C03624=1096.726,72.029,-58.754,176.200,16.216,152.221
C03625=1096.720,71.780,-58.738,176.198,16.216,152.221
C03626=1096.715,71.531,-58.720,176.195,16.215,152.221
C03627=1096.709,71.282,-58.704,176.193,16.214,152.222
C03628=1096.703,71.032,-58.687,176.190,16.213,152.222
C03629=1096.698,70.783,-58.670,176.188,16.213,152.222
C03630=1096.692,70.534,-58.654,176.185,16.211,152.223
C03631=1096.687,70.284,-58.637,176.183,16.211,152.223
C03632=1096.681,70.035,-58.620,176.180,16.210,152.223
C03633=1096.675,69.785,-58.602,176.179,16.209,152.224
C03634=1096.669,69.536,-58.586,176.176,16.209,152.224
C03635=1096.663,69.286,-58.569,176.174,16.208,152.224
C03636=1096.657,69.037,-58.552,176.172,16.207,152.225
C03637=1096.652,68.787,-58.536,176.169,16.206,152.225
C03638=1096.646,68.538,-58.519,176.167,16.205,152.225
C03639=1096.641,68.288,-58.502,176.164,16.205,152.226
C03640=1096.635,68.039,-58.486,176.162,16.204,152.226
C03641=1096.629,67.790,-58.469,176.159,16.203,152.226
C03642=1096.623,67.541,-58.452,176.157,16.202,152.227
C03643=1096.618,67.291,-58.436,176.155,16.201,152.227
C03644=1096.612,67.042,-58.419,176.152,16.201,152.227
C03645=1096.606,66.793,-58.402,176.150,16.200,152.228
C03646=1096.601,66.543,-58.385,176.148,16.199,152.228
C03647=1096.595,66.294,-58.369,176.146,16.199,152.228
C03648=1096.590,66.044,-58.352,176.143,16.197,152.228
C03649=1096.584,65.795,-58.336,176.141,16.197,152.229
C03650=1096.578,65.546,-58.320,176.138,16.196,152.229
C03651=1096.572,65.296,-58.303,176.136,16.195,152.229
C03652=1096.566,65.047,-58.286,176.133,16.194,152.230
C03653=1096.561,64.798,-58.269,176.131,16.194,152.230
C03654=1096.555,64.548,-58.253,176.129,16.192,152.230
C03655=1096.549,64.299,-58.237,176.127,16.192,152.231
C03656=1096.543,64.024,-58.218,176.124,16.191,152.231
C03657=1096.537,63.749,-58.200,176.122,16.190,152.231
C03658=1096.531,63.475,-58.182,176.119,16.189,152.232
C03659=1096.524,63.201,-58.164,176.116,16.188,152.232
C03660=1096.519,62.952,-58.147,176.114,16.187,152.232
C03661=1096.513,62.702,-58.131,176.111,16.186,152.233
C03662=1096.507,62.453,-58.115,176.109,16.186,152.233
C03663=1096.501,62.204,-58.098,176.107,16.185,152.233
C03664=1096.495,61.954,-58.082,176.105,16.184,152.234
C03665=1096.490,61.705,-58.065,176.103,16.184,152.234
C03666=1096.484,61.455,-58.049,176.100,16.182,152.234
C03667=1096.478,61.206,-58.033,176.098,16.182,152.235
C03668=1096.472,60.957,-58.017,176.095,16.181,152.235
C03669=1096.466,60.707,-58.000,176.093,16.180,152.235
C03670=1096.461,60.458,-57.983,176.091,16.179,152.235
C03671=1096.455,60.208,-57.967,176.088,16.179,152.236
C03672=1096.449,59.959,-57.951,176.086,16.178,152.236
C03673=1096.443,59.709,-57.935,176.084,16.177,152.236
C03674=1096.437,59.460,-57.918,176.082,16.176,152.237
C03675=1096.432,59.210,-57.902,176.079,16.175,152.237
C03676=1096.426,58.961,-57.885,176.077,16.174,152.237
C03677=1096.420,58.711,-57.870,176.075,16.174,152.238
C03678=1096.414,58.462,-57.854,176.072,16.172,152.238
C03679=1096.408,58.212,-57.837,176.070,16.172,152.238
C03680=1096.403,57.964,-57.821,176.068,16.171,152.239
C03681=1096.397,57.714,-57.805,176.066,16.170,152.239
C03682=1096.391,57.465,-57.788,176.063,16.169,152.239
C03683=1096.386,57.215,-57.772,176.061,16.168,152.239
C03684=1096.380,56.966,-57.756,176.059,16.168,152.240
C03685=1096.374,56.716,-57.740,176.056,16.167,152.240
C03686=1096.368,56.467,-57.724,176.054,16.166,152.240
C03687=1096.362,56.217,-57.708,176.052,16.165,152.240
C03688=1096.356,55.968,-57.691,176.050,16.164,152.241
C03689=1096.351,55.719,-57.675,176.048,16.163,152.241
C03690=1096.346,55.469,-57.659,176.045,16.162,152.241
C03691=1096.340,55.220,-57.643,176.043,16.161,152.242
C03692=1096.334,54.970,-57.627,176.040,16.161,152.242
C03693=1096.328,54.721,-57.611,176.038,16.160,152.242
C03694=1096.322,54.472,-57.594,176.036,16.159,152.242
C03695=1096.317,54.223,-57.579,176.034,16.158,152.243
C03696=1096.311,53.973,-57.563,176.032,16.157,152.243
C03697=1096.305,53.724,-57.547,176.029,16.156,152.243
C03698=1096.299,53.474,-57.531,176.027,16.155,152.244
C03699=1096.294,53.224,-57.514,176.025,16.154,152.244
C03700=1096.288,52.975,-57.498,176.023,16.153,152.244
C03701=1096.283,52.726,-57.482,176.021,16.153,152.244
C03702=1096.277,52.476,-57.467,176.018,16.151,152.245
C03703=1096.271,52.227,-57.450,176.016,16.151,152.245
C03704=1096.265,51.978,-57.434,176.014,16.149,152.245
C03705=1096.260,51.728,-57.419,176.011,16.149,152.246
C03706=1096.254,51.479,-57.403,176.010,16.148,152.246
C03707=1096.248,51.230,-57.386,176.007,16.147,152.246
C03708=1096.243,50.980,-57.371,176.005,16.146,152.246
C03709=1096.237,50.730,-57.355,176.002,16.145,152.247
C03710=1096.232,50.481,-57.339,176.000,16.144,152.247
C03711=1096.226,50.232,-57.323,175.999,16.144,152.247
C03712=1096.220,49.982,-57.307,175.996,16.142,152.247
C03713=1096.214,49.732,-57.291,175.994,16.142,152.248
C03714=1096.209,49.484,-57.276,175.991,16.140,152.248
C03715=1096.203,49.234,-57.260,175.989,16.140,152.248
C03716=1096.197,48.984,-57.244,175.988,16.139,152.248
C03717=1096.191,48.735,-57.227,175.985,16.137,152.249
C03718=1096.186,48.486,-57.212,175.983,16.137,152.249
C03719=1096.180,48.236,-57.196,175.981,16.135,152.249
C03720=1096.174,47.961,-57.178,175.979,16.135,152.249
C03721=1096.168,47.687,-57.161,175.976,16.133,152.250
C03722=1096.162,47.412,-57.143,175.973,16.132,152.250
C03723=1096.156,47.138,-57.127,175.971,16.131,152.250
C03724=1096.150,46.888,-57.111,175.969,16.130,152.250
C03725=1096.144,46.639,-57.095,175.967,16.129,152.251
C03726=1096.139,46.389,-57.079,175.965,16.129,152.251
C03727=1096.134,46.139,-57.064,175.962,16.127,152.251
C03728=1096.128,45.890,-57.048,175.960,16.127,152.251
C03729=1096.122,45.640,-57.032,175.958,16.125,152.252
C03730=1096.117,45.391,-57.016,175.956,16.125,152.252
C03731=1096.111,45.141,-57.001,175.954,16.124,152.252
C03732=1096.105,44.892,-56.985,175.951,16.122,152.252
C03733=1096.100,44.643,-56.969,175.950,16.122,152.253
C03734=1096.094,44.393,-56.953,175.948,16.121,152.253
C03735=1096.089,44.144,-56.938,175.945,16.120,152.253
C03736=1096.083,43.894,-56.922,175.943,16.119,152.253
C03737=1096.077,43.645,-56.906,175.940,16.118,152.254
C03738=1096.072,43.396,-56.891,175.939,16.117,152.254
C03739=1096.066,43.146,-56.876,175.937,16.116,152.254
C03740=1096.060,42.897,-56.860,175.934,16.115,152.254
C03741=1096.055,42.647,-56.845,175.932,16.114,152.255
C03742=1096.049,42.398,-56.828,175.930,16.112,152.255
C03743=1096.043,42.148,-56.813,175.928,16.112,152.255
C03744=1096.038,41.899,-56.798,175.926,16.111,152.255
C03745=1096.032,41.650,-56.782,175.923,16.110,152.256
C03746=1096.026,41.400,-56.766,175.921,16.109,152.256
C03747=1096.021,41.151,-56.751,175.919,16.108,152.256
C03748=1096.015,40.901,-56.736,175.917,16.107,152.256
C03749=1096.009,40.651,-56.720,175.915,16.106,152.256
C03750=1096.004,40.402,-56.705,175.913,16.105,152.257
C03751=1095.998,40.152,-56.689,175.911,16.104,152.257
C03752=1095.991,39.903,-56.674,175.909,16.103,152.257
C03753=1095.986,39.654,-56.658,175.906,16.102,152.258
C03754=1095.981,39.404,-56.643,175.904,16.101,152.258
C03755=1095.975,39.155,-56.628,175.903,16.100,152.258
C03756=1095.969,38.906,-56.612,175.900,16.099,152.258
C03757=1095.963,38.656,-56.597,175.898,16.098,152.258
C03758=1095.958,38.406,-56.581,175.896,16.098,152.259
C03759=1095.952,38.157,-56.566,175.893,16.096,152.259
C03760=1095.947,37.908,-56.551,175.892,16.095,152.259
C03761=1095.941,37.658,-56.535,175.890,16.094,152.259
C03762=1095.934,37.409,-56.520,175.887,16.093,152.260
C03763=1095.929,37.159,-56.505,175.885,16.092,152.260
C03764=1095.924,36.909,-56.489,175.883,16.091,152.260
C03765=1095.918,36.660,-56.475,175.881,16.090,152.260
C03766=1095.912,36.411,-56.459,175.879,16.089,152.260
C03767=1095.906,36.161,-56.444,175.876,16.088,152.261
C03768=1095.900,35.912,-56.428,175.875,16.087,152.261
C03769=1095.894,35.662,-56.413,175.873,16.087,152.261
C03770=1095.889,35.413,-56.398,175.870,16.085,152.262
C03771=1095.883,35.163,-56.383,175.868,16.084,152.262
C03772=1095.877,34.914,-56.368,175.866,16.083,152.262
C03773=1095.872,34.664,-56.353,175.864,16.082,152.262
C03774=1095.866,34.415,-56.338,175.862,16.081,152.262
C03775=1095.860,34.166,-56.322,175.860,16.081,152.263
C03776=1095.854,33.916,-56.307,175.858,16.079,152.263
C03777=1095.849,33.667,-56.292,175.856,16.078,152.263
C03778=1095.842,33.417,-56.277,175.854,16.078,152.263
C03779=1095.837,33.167,-56.261,175.851,16.076,152.264
C03780=1095.831,32.918,-56.247,175.850,16.075,152.264
C03781=1095.825,32.668,-56.231,175.848,16.074,152.264
C03782=1095.820,32.419,-56.216,175.845,16.073,152.264
C03783=1095.814,32.170,-56.201,175.843,16.073,152.265
C03784=1095.808,31.895,-56.185,175.841,16.071,152.265
C03785=1095.802,31.621,-56.168,175.839,16.070,152.265
C03786=1095.795,31.345,-56.151,175.836,16.069,152.265
C03787=1095.789,31.071,-56.134,175.834,16.068,152.265
C03788=1095.783,30.822,-56.120,175.832,16.066,152.266
C03789=1095.778,30.572,-56.104,175.830,16.066,152.266
C03790=1095.771,30.323,-56.089,175.828,16.065,152.266
C03791=1095.766,30.073,-56.074,175.825,16.064,152.266
C03792=1095.760,29.824,-56.059,175.824,16.063,152.266
C03793=1095.755,29.574,-56.045,175.822,16.062,152.267
C03794=1095.749,29.324,-56.030,175.819,16.061,152.267
C03795=1095.744,29.075,-56.015,175.818,16.059,152.267
C03796=1095.738,28.826,-56.000,175.816,16.059,152.267
C03797=1095.732,28.576,-55.985,175.813,16.057,152.268
C03798=1095.727,28.327,-55.970,175.811,16.056,152.268
C03799=1095.720,28.077,-55.955,175.810,16.056,152.268
C03800=1095.715,27.828,-55.940,175.807,16.054,152.268
C03801=1095.709,27.578,-55.925,175.805,16.053,152.268
C03802=1095.703,27.329,-55.911,175.803,16.052,152.269
C03803=1095.698,27.079,-55.896,175.801,16.051,152.269
C03804=1095.692,26.830,-55.881,175.799,16.050,152.269
C03805=1095.686,26.580,-55.865,175.797,16.049,152.269
C03806=1095.680,26.331,-55.851,175.795,16.048,152.270
C03807=1095.674,26.081,-55.836,175.793,16.047,152.270
C03808=1095.668,25.832,-55.821,175.791,16.046,152.270
C03809=1095.663,25.582,-55.806,175.789,16.045,152.270
C03810=1095.657,25.333,-55.792,175.787,16.044,152.270
C03811=1095.651,25.083,-55.777,175.785,16.043,152.270
C03812=1095.646,24.834,-55.762,175.783,16.042,152.271
C03813=1095.640,24.584,-55.748,175.781,16.041,152.271
C03814=1095.634,24.335,-55.733,175.779,16.040,152.271
C03815=1095.629,24.085,-55.718,175.777,16.039,152.271
C03816=1095.622,23.836,-55.703,175.774,16.037,152.272
C03817=1095.617,23.586,-55.689,175.773,16.037,152.272
C03818=1095.611,23.337,-55.674,175.771,16.036,152.272
C03819=1095.605,23.087,-55.659,175.768,16.034,152.272
C03820=1095.599,22.838,-55.644,175.766,16.034,152.272
C03821=1095.594,22.588,-55.630,175.765,16.032,152.272
C03822=1095.589,22.339,-55.615,175.763,16.032,152.273
C03823=1095.582,22.089,-55.600,175.760,16.030,152.273
C03824=1095.577,21.840,-55.586,175.759,16.029,152.273
C03825=1095.570,21.590,-55.571,175.757,16.029,152.273
C03826=1095.565,21.341,-55.556,175.754,16.027,152.274
C03827=1095.560,21.091,-55.542,175.752,16.026,152.274
C03828=1095.553,20.841,-55.527,175.751,16.025,152.274
C03829=1095.548,20.592,-55.513,175.748,16.024,152.274
C03830=1095.543,20.343,-55.498,175.746,16.023,152.274
C03831=1095.537,20.093,-55.483,175.745,16.022,152.275
C03832=1095.531,19.844,-55.469,175.743,16.021,152.275
C03833=1095.525,19.594,-55.454,175.740,16.020,152.275
C03834=1095.519,19.345,-55.440,175.738,16.019,152.275
C03835=1095.513,19.095,-55.426,175.737,16.018,152.275
C03836=1095.507,18.845,-55.411,175.734,16.016,152.276
C03837=1095.502,18.596,-55.396,175.732,16.016,152.276
C03838=1095.497,18.347,-55.382,175.731,16.014,152.276
C03839=1095.490,18.097,-55.367,175.729,16.014,152.276
C03840=1095.485,17.847,-55.353,175.726,16.012,152.276
C03841=1095.479,17.598,-55.339,175.725,16.011,152.277
C03842=1095.473,17.348,-55.324,175.723,16.011,152.277
C03843=1095.467,17.099,-55.310,175.720,16.009,152.277
C03844=1095.462,16.850,-55.295,175.718,16.008,152.277
C03845=1095.456,16.600,-55.280,175.717,16.007,152.277
C03846=1095.450,16.351,-55.266,175.715,16.006,152.277
C03847=1095.445,16.101,-55.252,175.712,16.004,152.278
C03848=1095.438,15.827,-55.236,175.711,16.004,152.278
C03849=1095.431,15.554,-55.220,175.708,16.003,152.278
C03850=1095.425,15.281,-55.204,175.706,16.001,152.278
C03851=1095.419,15.008,-55.188,175.704,16.000,152.279
C03852=1095.413,14.758,-55.175,175.702,15.999,152.279
C03853=1095.408,14.509,-55.160,175.700,15.998,152.279
C03854=1095.402,14.259,-55.146,175.699,15.997,152.279
C03855=1095.396,14.010,-55.131,175.696,15.996,152.279
C03856=1095.390,13.760,-55.117,175.694,15.995,152.279
C03857=1095.384,13.511,-55.102,175.692,15.994,152.280
C03858=1095.378,13.261,-55.089,175.690,15.993,152.280
C03859=1095.373,13.012,-55.074,175.688,15.991,152.280
C03860=1095.367,12.762,-55.060,175.686,15.991,152.280
C03861=1095.361,12.512,-55.046,175.685,15.990,152.280
C03862=1095.355,12.263,-55.031,175.683,15.989,152.281
C03863=1095.349,12.013,-55.018,175.680,15.987,152.281
C03864=1095.343,11.764,-55.004,175.678,15.986,152.281
C03865=1095.337,11.515,-54.989,175.677,15.986,152.281
C03866=1095.332,11.265,-54.975,175.674,15.984,152.281
C03867=1095.325,11.015,-54.960,175.672,15.983,152.282
C03868=1095.320,10.766,-54.947,175.671,15.982,152.282
C03869=1095.314,10.516,-54.933,175.669,15.981,152.282
C03870=1095.308,10.267,-54.918,175.666,15.980,152.282
C03871=1095.303,10.017,-54.904,175.664,15.979,152.282
C03872=1095.297,9.767,-54.890,175.663,15.978,152.282
C03873=1095.291,9.519,-54.876,175.661,15.977,152.283
C03874=1095.285,9.269,-54.862,175.659,15.975,152.283
C03875=1095.279,9.019,-54.848,175.657,15.975,152.283
C03876=1095.274,8.769,-54.834,175.655,15.974,152.283
C03877=1095.268,8.520,-54.819,175.653,15.973,152.283
C03878=1095.262,8.270,-54.805,175.651,15.971,152.284
C03879=1095.256,8.021,-54.791,175.649,15.970,152.284
C03880=1095.250,7.771,-54.778,175.647,15.969,152.284
C03881=1095.244,7.522,-54.764,175.645,15.969,152.284
C03882=1095.238,7.272,-54.749,175.644,15.967,152.284
C03883=1095.233,7.023,-54.735,175.641,15.966,152.285
C03884=1095.227,6.773,-54.722,175.640,15.965,152.285
C03885=1095.221,6.524,-54.707,175.638,15.964,152.285
C03886=1095.216,6.274,-54.693,175.636,15.963,152.285
C03887=1095.209,6.024,-54.680,175.634,15.961,152.285
C03888=1095.204,5.775,-54.666,175.632,15.961,152.285
C03889=1095.198,5.525,-54.652,175.630,15.959,152.286
C03890=1095.192,5.276,-54.637,175.628,15.959,152.286
C03891=1095.187,5.027,-54.623,175.626,15.957,152.286
C03892=1095.180,4.777,-54.610,175.624,15.956,152.286
C03893=1095.175,4.527,-54.596,175.622,15.955,152.286
C03894=1095.169,4.278,-54.582,175.621,15.954,152.287
C03895=1095.164,4.028,-54.568,175.618,15.953,152.287
C03896=1095.158,3.779,-54.554,175.617,15.952,152.287
C03897=1095.152,3.529,-54.541,175.615,15.951,152.287
C03898=1095.146,3.280,-54.526,175.613,15.950,152.287
C03899=1095.140,3.030,-54.512,175.610,15.948,152.287
C03900=1095.135,2.780,-54.498,175.609,15.947,152.288
C03901=1095.129,2.531,-54.484,175.607,15.946,152.288
C03902=1095.123,2.282,-54.471,175.605,15.945,152.288
C03903=1095.118,2.032,-54.457,175.604,15.944,152.288
C03904=1095.112,1.782,-54.443,175.601,15.943,152.288
C03905=1095.106,1.532,-54.429,175.599,15.942,152.288
C03906=1095.100,1.283,-54.415,175.598,15.941,152.288
C03907=1095.094,1.033,-54.402,175.596,15.940,152.289
C03908=1095.089,0.784,-54.388,175.594,15.938,152.289
C03909=1095.083,0.534,-54.374,175.592,15.937,152.289
C03910=1095.078,0.285,-54.360,175.590,15.936,152.289
C03911=1095.072,0.035,-54.347,175.589,15.935,152.289
C03912=1095.065,-0.236,-54.332,175.586,15.934,152.290
C03913=1095.059,-0.507,-54.317,175.584,15.933,152.290
C03914=1095.053,-0.779,-54.302,175.582,15.932,152.290
C03915=1095.047,-1.049,-54.287,175.580,15.930,152.290
C03916=1095.041,-1.299,-54.273,175.578,15.929,152.290
C03917=1095.035,-1.548,-54.260,175.576,15.928,152.290
C03918=1095.029,-1.799,-54.246,175.575,15.927,152.291
C03919=1095.024,-2.048,-54.232,175.572,15.925,152.291
C03920=1095.018,-2.298,-54.219,175.571,15.925,152.291
C03921=1095.012,-2.548,-54.205,175.569,15.924,152.291
C03922=1095.007,-2.797,-54.192,175.567,15.922,152.291
C03923=1095.001,-3.047,-54.178,175.565,15.921,152.291
C03924=1094.995,-3.296,-54.164,175.563,15.920,152.292
C03925=1094.990,-3.546,-54.151,175.562,15.919,152.292
C03926=1094.984,-3.795,-54.137,175.560,15.918,152.292
C03927=1094.978,-4.044,-54.123,175.558,15.917,152.292
C03928=1094.972,-4.294,-54.110,175.555,15.916,152.292
C03929=1094.966,-4.543,-54.096,175.554,15.915,152.292
C03930=1094.961,-4.793,-54.083,175.552,15.914,152.293
C03931=1094.954,-5.043,-54.069,175.550,15.913,152.293
C03932=1094.949,-5.293,-54.056,175.549,15.912,152.293
C03933=1094.943,-5.542,-54.042,175.546,15.910,152.293
C03934=1094.937,-5.792,-54.028,175.544,15.909,152.293
C03935=1094.931,-6.041,-54.015,175.543,15.908,152.293
C03936=1094.925,-6.291,-54.001,175.541,15.907,152.294
C03937=1094.919,-6.541,-53.989,175.539,15.906,152.294
C03938=1094.914,-6.790,-53.975,175.537,15.905,152.294
C03939=1094.908,-7.039,-53.962,175.535,15.904,152.294
C03940=1094.902,-7.289,-53.948,175.533,15.903,152.294
C03941=1094.896,-7.538,-53.935,175.532,15.902,152.294
C03942=1094.890,-7.788,-53.922,175.530,15.901,152.294
C03943=1094.885,-8.038,-53.908,175.528,15.900,152.295
C03944=1094.878,-8.287,-53.895,175.526,15.898,152.295
C03945=1094.873,-8.536,-53.881,175.524,15.897,152.295
C03946=1094.867,-8.786,-53.868,175.522,15.896,152.295
C03947=1094.862,-9.036,-53.855,175.521,15.895,152.295
C03948=1094.855,-9.285,-53.841,175.519,15.894,152.296
C03949=1094.850,-9.535,-53.827,175.517,15.893,152.296
C03950=1094.844,-9.785,-53.815,175.515,15.892,152.296
C03951=1094.838,-10.034,-53.802,175.513,15.891,152.296
C03952=1094.832,-10.284,-53.788,175.511,15.890,152.296
C03953=1094.826,-10.533,-53.775,175.510,15.888,152.296
C03954=1094.821,-10.783,-53.761,175.508,15.888,152.297
C03955=1094.815,-11.032,-53.748,175.505,15.886,152.297
C03956=1094.810,-11.282,-53.735,175.504,15.885,152.297
C03957=1094.803,-11.532,-53.722,175.502,15.884,152.297
C03958=1094.797,-11.781,-53.708,175.500,15.883,152.297
C03959=1094.792,-12.031,-53.695,175.499,15.882,152.297
C03960=1094.786,-12.280,-53.682,175.497,15.881,152.297
C03961=1094.780,-12.530,-53.668,175.494,15.879,152.298
C03962=1094.774,-12.780,-53.656,175.493,15.878,152.298
C03963=1094.768,-13.029,-53.642,175.491,15.878,152.298
C03964=1094.763,-13.279,-53.628,175.489,15.876,152.298
C03965=1094.757,-13.529,-53.616,175.488,15.875,152.298
C03966=1094.751,-13.778,-53.602,175.486,15.875,152.298
C03967=1094.745,-14.028,-53.589,175.483,15.873,152.299
C03968=1094.739,-14.277,-53.576,175.482,15.872,152.299
C03969=1094.734,-14.527,-53.562,175.480,15.871,152.299
C03970=1094.728,-14.777,-53.550,175.478,15.870,152.299
C03971=1094.722,-15.026,-53.536,175.477,15.869,152.299
C03972=1094.716,-15.276,-53.523,175.475,15.868,152.299
C03973=1094.710,-15.526,-53.510,175.473,15.867,152.299
C03974=1094.704,-15.775,-53.497,175.471,15.865,152.300
C03975=1094.698,-16.025,-53.484,175.469,15.864,152.300
C03976=1094.692,-16.294,-53.470,175.467,15.863,152.300
C03977=1094.686,-16.563,-53.456,175.466,15.862,152.300
C03978=1094.680,-16.834,-53.442,175.463,15.861,152.300
C03979=1094.674,-17.103,-53.428,175.462,15.860,152.300
C03980=1094.667,-17.353,-53.415,175.460,15.859,152.301
C03981=1094.662,-17.602,-53.402,175.458,15.858,152.301
C03982=1094.655,-17.852,-53.389,175.456,15.856,152.301
C03983=1094.650,-18.102,-53.376,175.454,15.855,152.301
C03984=1094.644,-18.351,-53.362,175.452,15.854,152.301
C03985=1094.638,-18.601,-53.350,175.451,15.853,152.301
C03986=1094.632,-18.850,-53.337,175.449,15.852,152.302
C03987=1094.626,-19.099,-53.324,175.447,15.851,152.302
C03988=1094.620,-19.349,-53.311,175.445,15.850,152.302
C03989=1094.615,-19.599,-53.298,175.444,15.849,152.302
C03990=1094.609,-19.849,-53.285,175.441,15.847,152.302
C03991=1094.603,-20.098,-53.272,175.439,15.847,152.303
C03992=1094.597,-20.348,-53.260,175.438,15.846,152.303
C03993=1094.591,-20.597,-53.246,175.436,15.844,152.303
C03994=1094.585,-20.847,-53.234,175.434,15.844,152.303
C03995=1094.580,-21.097,-53.221,175.433,15.843,152.303
C03996=1094.574,-21.346,-53.208,175.431,15.841,152.303
C03997=1094.568,-21.596,-53.195,175.429,15.841,152.303
C03998=1094.562,-21.845,-53.182,175.427,15.839,152.304
C03999=1094.556,-22.095,-53.169,175.425,15.838,152.304
C04000=1094.550,-22.345,-53.157,175.424,15.837,152.304
C04001=1094.545,-22.594,-53.143,175.422,15.836,152.304
C04002=1094.539,-22.844,-53.130,175.420,15.835,152.304
C04003=1094.534,-23.093,-53.118,175.419,15.834,152.304
C04004=1094.527,-23.343,-53.105,175.417,15.833,152.304
C04005=1094.521,-23.593,-53.092,175.415,15.832,152.305
C04006=1094.516,-23.842,-53.080,175.413,15.830,152.305
C04007=1094.509,-24.092,-53.067,175.411,15.829,152.305
C04008=1094.503,-24.342,-53.054,175.409,15.828,152.305
C04009=1094.498,-24.591,-53.042,175.408,15.827,152.305
C04010=1094.493,-24.841,-53.029,175.406,15.826,152.305
C04011=1094.487,-25.090,-53.015,175.404,15.825,152.306
C04012=1094.481,-25.340,-53.003,175.403,15.824,152.306
C04013=1094.475,-25.590,-52.990,175.401,15.823,152.306
C04014=1094.470,-25.839,-52.978,175.398,15.821,152.306
C04015=1094.463,-26.088,-52.965,175.397,15.820,152.306
C04016=1094.457,-26.338,-52.952,175.395,15.819,152.306
C04017=1094.452,-26.588,-52.940,175.393,15.818,152.306
C04018=1094.446,-26.838,-52.927,175.392,15.817,152.307
C04019=1094.440,-27.087,-52.914,175.390,15.816,152.307
C04020=1094.434,-27.337,-52.902,175.388,15.815,152.307
C04021=1094.428,-27.586,-52.889,175.386,15.814,152.307
C04022=1094.422,-27.836,-52.877,175.385,15.813,152.307
C04023=1094.416,-28.086,-52.864,175.383,15.812,152.307
C04024=1094.411,-28.335,-52.851,175.381,15.811,152.308
C04025=1094.405,-28.585,-52.839,175.379,15.809,152.308
C04026=1094.399,-28.835,-52.826,175.377,15.809,152.308
C04027=1094.393,-29.084,-52.813,175.376,15.808,152.308
C04028=1094.387,-29.334,-52.801,175.374,15.806,152.308
C04029=1094.382,-29.583,-52.789,175.372,15.806,152.308
C04030=1094.375,-29.832,-52.776,175.370,15.805,152.308
C04031=1094.369,-30.082,-52.763,175.369,15.804,152.309
C04032=1094.363,-30.332,-52.751,175.367,15.803,152.309
C04033=1094.357,-30.582,-52.738,175.365,15.802,152.309
C04034=1094.352,-30.831,-52.726,175.363,15.801,152.309
C04035=1094.346,-31.081,-52.714,175.361,15.799,152.309
C04036=1094.340,-31.331,-52.701,175.360,15.798,152.309
C04037=1094.334,-31.581,-52.689,175.358,15.797,152.310
C04038=1094.329,-31.829,-52.676,175.356,15.796,152.310
C04039=1094.323,-32.079,-52.663,175.354,15.795,152.310
C04040=1094.316,-32.349,-52.650,175.353,15.794,152.310
C04041=1094.310,-32.617,-52.637,175.351,15.793,152.310
C04042=1094.303,-32.886,-52.624,175.349,15.791,152.310
C04043=1094.297,-33.155,-52.610,175.347,15.791,152.311
C04044=1094.291,-33.404,-52.598,175.345,15.790,152.311
C04045=1094.285,-33.654,-52.585,175.343,15.788,152.311
C04046=1094.279,-33.904,-52.573,175.342,15.788,152.311
C04047=1094.274,-34.153,-52.560,175.340,15.787,152.311
C04048=1094.267,-34.403,-52.548,175.338,15.785,152.311
C04049=1094.261,-34.653,-52.536,175.336,15.785,152.312
C04050=1094.256,-34.902,-52.524,175.335,15.783,152.312
C04051=1094.250,-35.152,-52.511,175.333,15.782,152.312
C04052=1094.244,-35.402,-52.499,175.331,15.782,152.312
C04053=1094.239,-35.651,-52.486,175.330,15.780,152.312
C04054=1094.232,-35.901,-52.474,175.327,15.779,152.312
C04055=1094.226,-36.150,-52.462,175.326,15.778,152.313
C04056=1094.221,-36.400,-52.449,175.324,15.777,152.313
C04057=1094.215,-36.650,-52.437,175.322,15.776,152.313
C04058=1094.209,-36.899,-52.425,175.321,15.775,152.313
C04059=1094.203,-37.149,-52.412,175.319,15.774,152.313
C04060=1094.197,-37.398,-52.400,175.317,15.773,152.313
C04061=1094.191,-37.648,-52.388,175.316,15.772,152.313
C04062=1094.186,-37.897,-52.376,175.314,15.771,152.314
C04063=1094.180,-38.147,-52.363,175.312,15.770,152.314
C04064=1094.175,-38.398,-52.351,175.311,15.768,152.314
C04065=1094.169,-38.646,-52.340,175.309,15.768,152.314
C04066=1094.163,-38.896,-52.327,175.307,15.767,152.314
C04067=1094.157,-39.146,-52.315,175.306,15.765,152.314
C04068=1094.150,-39.396,-52.303,175.304,15.765,152.314
C04069=1094.145,-39.645,-52.290,175.302,15.764,152.315
C04070=1094.139,-39.895,-52.278,175.300,15.762,152.315
C04071=1094.132,-40.144,-52.266,175.299,15.762,152.315
C04072=1094.127,-40.394,-52.254,175.297,15.761,152.315
C04073=1094.121,-40.644,-52.242,175.295,15.760,152.315
C04074=1094.115,-40.894,-52.230,175.293,15.758,152.315
C04075=1094.109,-41.143,-52.218,175.291,15.757,152.316
C04076=1094.103,-41.392,-52.206,175.289,15.756,152.316
C04077=1094.097,-41.642,-52.193,175.288,15.755,152.316
C04078=1094.092,-41.892,-52.182,175.286,15.754,152.316
C04079=1094.085,-42.142,-52.170,175.284,15.753,152.316
C04080=1094.079,-42.392,-52.157,175.283,15.752,152.316
C04081=1094.074,-42.641,-52.145,175.281,15.751,152.317
C04082=1094.067,-42.890,-52.133,175.279,15.750,152.317
C04083=1094.062,-43.140,-52.122,175.277,15.749,152.317
C04084=1094.056,-43.390,-52.110,175.276,15.748,152.317
C04085=1094.050,-43.640,-52.097,175.274,15.747,152.317
C04086=1094.044,-43.889,-52.085,175.272,15.746,152.317
C04087=1094.038,-44.139,-52.074,175.270,15.745,152.318
C04088=1094.032,-44.389,-52.061,175.269,15.744,152.318
C04089=1094.026,-44.638,-52.050,175.267,15.743,152.318
C04090=1094.020,-44.888,-52.037,175.265,15.742,152.318
C04091=1094.015,-45.137,-52.026,175.264,15.741,152.318
C04092=1094.009,-45.387,-52.014,175.262,15.740,152.318
C04093=1094.003,-45.637,-52.001,175.260,15.739,152.318
C04094=1093.997,-45.886,-51.990,175.259,15.738,152.319
C04095=1093.991,-46.136,-51.978,175.257,15.738,152.319
C04096=1093.985,-46.385,-51.966,175.255,15.736,152.319
C04097=1093.979,-46.635,-51.953,175.254,15.735,152.319
C04098=1093.973,-46.884,-51.943,175.252,15.735,152.319
C04099=1093.967,-47.134,-51.930,175.250,15.733,152.319
C04100=1093.962,-47.384,-51.917,175.249,15.732,152.320
C04101=1093.956,-47.634,-51.907,175.247,15.732,152.320
C04102=1093.950,-47.884,-51.894,175.245,15.730,152.320
C04103=1093.944,-48.133,-51.883,175.243,15.729,152.320
C04104=1093.938,-48.402,-51.870,175.242,15.729,152.320
C04105=1093.932,-48.671,-51.857,175.240,15.727,152.320
C04106=1093.925,-48.940,-51.844,175.237,15.726,152.321
C04107=1093.919,-49.210,-51.832,175.236,15.725,152.321
C04108=1093.913,-49.459,-51.820,175.234,15.724,152.321
C04109=1093.908,-49.709,-51.808,175.232,15.723,152.321
C04110=1093.901,-49.959,-51.796,175.231,15.722,152.321
C04111=1093.895,-50.208,-51.784,175.229,15.721,152.321
C04112=1093.889,-50.458,-51.773,175.227,15.720,152.322
C04113=1093.883,-50.708,-51.760,175.226,15.719,152.322
C04114=1093.878,-50.957,-51.749,175.224,15.718,152.322
C04115=1093.871,-51.207,-51.738,175.222,15.717,152.322
C04116=1093.866,-51.457,-51.726,175.220,15.716,152.322
C04117=1093.859,-51.706,-51.714,175.219,15.715,152.322
C04118=1093.853,-51.956,-51.702,175.217,15.714,152.323
C04119=1093.848,-52.206,-51.691,175.215,15.713,152.323
C04120=1093.841,-52.455,-51.679,175.213,15.712,152.323
C04121=1093.835,-52.705,-51.668,175.212,15.712,152.323
C04122=1093.829,-52.954,-51.656,175.211,15.711,152.323
C04123=1093.824,-53.204,-51.644,175.209,15.710,152.323
C04124=1093.817,-53.454,-51.632,175.207,15.709,152.324
C04125=1093.811,-53.704,-51.621,175.205,15.708,152.324
C04126=1093.805,-53.953,-51.610,175.204,15.707,152.324
C04127=1093.799,-54.203,-51.598,175.202,15.706,152.324
C04128=1093.793,-54.452,-51.586,175.200,15.705,152.324
C04129=1093.787,-54.702,-51.575,175.199,15.704,152.324
C04130=1093.781,-54.951,-51.563,175.197,15.704,152.325
C04131=1093.775,-55.202,-51.551,175.195,15.702,152.325
C04132=1093.769,-55.450,-51.540,175.193,15.702,152.325
C04133=1093.763,-55.701,-51.529,175.192,15.701,152.325
C04134=1093.758,-55.950,-51.517,175.190,15.700,152.325
C04135=1093.751,-56.200,-51.505,175.188,15.699,152.325
C04136=1093.745,-56.450,-51.494,175.186,15.698,152.326
C04137=1093.739,-56.699,-51.482,175.185,15.697,152.326
C04138=1093.732,-56.949,-51.471,175.183,15.696,152.326
C04139=1093.727,-57.198,-51.459,175.181,15.695,152.326
C04140=1093.721,-57.449,-51.448,175.180,15.694,152.326
C04141=1093.715,-57.698,-51.437,175.178,15.693,152.327
C04142=1093.708,-57.948,-51.425,175.176,15.692,152.327
C04143=1093.703,-58.198,-51.413,175.174,15.691,152.327
C04144=1093.697,-58.447,-51.403,175.173,15.690,152.327
C04145=1093.691,-58.697,-51.391,175.172,15.690,152.327
C04146=1093.685,-58.946,-51.380,175.170,15.689,152.327
C04147=1093.678,-59.196,-51.368,175.168,15.688,152.328
C04148=1093.673,-59.445,-51.356,175.167,15.687,152.328
C04149=1093.667,-59.696,-51.345,175.165,15.686,152.328
C04150=1093.661,-59.945,-51.333,175.163,15.685,152.328
C04151=1093.655,-60.195,-51.322,175.161,15.684,152.328
C04152=1093.649,-60.444,-51.311,175.160,15.683,152.328
C04153=1093.643,-60.694,-51.299,175.158,15.682,152.329
C04154=1093.637,-60.944,-51.288,175.156,15.682,152.329
C04155=1093.631,-61.194,-51.277,175.154,15.680,152.329
C04156=1093.625,-61.443,-51.266,175.153,15.680,152.329
C04157=1093.619,-61.692,-51.254,175.151,15.679,152.329
C04158=1093.613,-61.942,-51.243,175.149,15.678,152.330
C04159=1093.608,-62.192,-51.231,175.147,15.677,152.330
C04160=1093.601,-62.442,-51.220,175.147,15.676,152.330
C04161=1093.595,-62.691,-51.209,175.145,15.675,152.330
C04162=1093.589,-62.941,-51.197,175.143,15.674,152.330
C04163=1093.583,-63.191,-51.186,175.141,15.674,152.330
C04164=1093.578,-63.440,-51.176,175.140,15.672,152.330
C04165=1093.572,-63.690,-51.163,175.138,15.672,152.331
C04166=1093.566,-63.940,-51.152,175.136,15.671,152.331
C04167=1093.560,-64.189,-51.141,175.134,15.670,152.331
C04168=1093.554,-64.460,-51.129,175.133,15.669,152.331
C04169=1093.547,-64.730,-51.117,175.131,15.668,152.331
C04170=1093.541,-65.001,-51.104,175.129,15.667,152.332
C04171=1093.534,-65.271,-51.093,175.127,15.666,152.332
C04172=1093.529,-65.521,-51.081,175.126,15.665,152.332
C04173=1093.522,-65.771,-51.070,175.124,15.664,152.332
C04174=1093.516,-66.020,-51.058,175.122,15.663,152.332
C04175=1093.511,-66.270,-51.047,175.120,15.663,152.333
C04176=1093.504,-66.520,-51.036,175.119,15.661,152.333
C04177=1093.498,-66.769,-51.025,175.117,15.661,152.333
C04178=1093.493,-67.019,-51.014,175.115,15.660,152.333
C04179=1093.486,-67.269,-51.003,175.114,15.659,152.333
C04180=1093.481,-67.519,-50.992,175.113,15.658,152.333
C04181=1093.475,-67.768,-50.980,175.111,15.657,152.333
C04182=1093.469,-68.018,-50.969,175.109,15.656,152.334
C04183=1093.463,-68.267,-50.958,175.108,15.655,152.334
C04184=1093.457,-68.517,-50.947,175.106,15.655,152.334
C04185=1093.451,-68.767,-50.936,175.104,15.653,152.334
C04186=1093.445,-69.017,-50.925,175.102,15.653,152.334
C04187=1093.440,-69.266,-50.914,175.101,15.652,152.335
C04188=1093.433,-69.516,-50.903,175.099,15.652,152.335
C04189=1093.428,-69.766,-50.892,175.098,15.650,152.335
C04190=1093.422,-70.015,-50.881,175.096,15.650,152.335
C04191=1093.416,-70.265,-50.870,175.094,15.649,152.335
C04192=1093.410,-70.515,-50.859,175.092,15.648,152.336
C04193=1093.404,-70.764,-50.848,175.091,15.647,152.336
C04194=1093.399,-71.014,-50.836,175.089,15.646,152.336
C04195=1093.392,-71.264,-50.825,175.087,15.645,152.336
C04196=1093.387,-71.513,-50.814,175.086,15.644,152.336
C04197=1093.381,-71.763,-50.803,175.085,15.644,152.336
C04198=1093.375,-72.012,-50.792,175.083,15.642,152.336
C04199=1093.369,-72.262,-50.781,175.081,15.642,152.337
C04200=1093.363,-72.512,-50.770,175.080,15.641,152.337
C04201=1093.357,-72.761,-50.759,175.078,15.640,152.337
C04202=1093.352,-73.011,-50.748,175.076,15.639,152.337
C04203=1093.345,-73.261,-50.737,175.074,15.638,152.337
C04204=1093.340,-73.511,-50.727,175.073,15.637,152.338
C04205=1093.334,-73.761,-50.716,175.072,15.637,152.338
C04206=1093.328,-74.010,-50.705,175.070,15.636,152.338
C04207=1093.322,-74.260,-50.694,175.068,15.635,152.338
C04208=1093.316,-74.510,-50.683,175.066,15.634,152.338
C04209=1093.311,-74.759,-50.672,175.065,15.633,152.338
C04210=1093.305,-75.009,-50.661,175.063,15.632,152.339
C04211=1093.298,-75.259,-50.650,175.061,15.631,152.339
C04212=1093.292,-75.508,-50.640,175.060,15.631,152.339
C04213=1093.286,-75.758,-50.629,175.058,15.630,152.339
C04214=1093.280,-76.008,-50.617,175.056,15.629,152.339
C04215=1093.274,-76.257,-50.607,175.055,15.628,152.340
C04216=1093.268,-76.507,-50.596,175.053,15.628,152.340
C04217=1093.263,-76.756,-50.585,175.051,15.627,152.340
C04218=1093.256,-77.006,-50.574,175.049,15.626,152.340
C04219=1093.250,-77.256,-50.564,175.048,15.626,152.340
C04220=1093.244,-77.506,-50.553,175.047,15.624,152.341
C04221=1093.239,-77.755,-50.542,175.045,15.624,152.341
C04222=1093.232,-78.006,-50.531,175.043,15.623,152.341
C04223=1093.226,-78.255,-50.521,175.041,15.622,152.341
C04224=1093.220,-78.504,-50.510,175.039,15.621,152.341
C04225=1093.214,-78.754,-50.499,175.039,15.621,152.341
C04226=1093.208,-79.005,-50.488,175.037,15.620,152.342
C04227=1093.203,-79.254,-50.478,175.035,15.619,152.342
C04228=1093.197,-79.503,-50.467,175.033,15.618,152.342
C04229=1093.190,-79.753,-50.456,175.031,15.618,152.342
C04230=1093.184,-80.003,-50.445,175.030,15.616,152.342
C04231=1093.178,-80.252,-50.434,175.029,15.616,152.343
C04232=1093.172,-80.525,-50.423,175.027,15.616,152.343
C04233=1093.165,-80.798,-50.412,175.025,15.614,152.343
C04234=1093.158,-81.071,-50.400,175.023,15.614,152.343
C04235=1093.152,-81.343,-50.388,175.021,15.613,152.344
C04236=1093.146,-81.593,-50.378,175.020,15.612,152.344
C04237=1093.139,-81.843,-50.367,175.018,15.611,152.344
C04238=1093.133,-82.092,-50.356,175.016,15.611,152.344
C04239=1093.128,-82.342,-50.346,175.014,15.610,152.345
C04240=1093.121,-82.591,-50.335,175.013,15.609,152.345
C04241=1093.115,-82.842,-50.325,175.011,15.609,152.345
C04242=1093.109,-83.091,-50.314,175.010,15.608,152.345
C04243=1093.103,-83.340,-50.304,175.008,15.607,152.345
C04244=1093.097,-83.590,-50.293,175.006,15.606,152.345
C04245=1093.090,-83.840,-50.283,175.005,15.606,152.346
C04246=1093.085,-84.090,-50.272,175.003,15.605,152.346
C04247=1093.079,-84.339,-50.261,175.001,15.604,152.346
C04248=1093.073,-84.589,-50.252,175.000,15.604,152.346
C04249=1093.067,-84.839,-50.241,174.998,15.602,152.346
C04250=1093.061,-85.089,-50.229,174.997,15.602,152.347
C04251=1093.054,-85.338,-50.219,174.995,15.602,152.347
C04252=1093.049,-85.588,-50.209,174.993,15.600,152.347
C04253=1093.042,-85.837,-50.199,174.991,15.600,152.347
C04254=1093.037,-86.087,-50.188,174.990,15.600,152.347
C04255=1093.031,-86.338,-50.177,174.988,15.599,152.348
C04256=1093.024,-86.587,-50.167,174.987,15.598,152.348
C04257=1093.018,-86.836,-50.156,174.985,15.597,152.348
C04258=1093.012,-87.086,-50.147,174.983,15.597,152.348
C04259=1093.006,-87.336,-50.136,174.982,15.596,152.348
C04260=1093.000,-87.586,-50.126,174.980,15.595,152.349
C04261=1092.994,-87.836,-50.115,174.978,15.595,152.349
C04262=1092.988,-88.085,-50.104,174.977,15.593,152.349
C04263=1092.982,-88.335,-50.094,174.975,15.593,152.349
C04264=1092.976,-88.584,-50.084,174.974,15.593,152.350
C04265=1092.970,-88.833,-50.073,174.972,15.592,152.350
C04266=1092.964,-89.084,-50.063,174.970,15.591,152.350
C04267=1092.957,-89.333,-50.052,174.968,15.590,152.350
C04268=1092.952,-89.584,-50.042,174.967,15.590,152.350
C04269=1092.946,-89.833,-50.031,174.966,15.589,152.351
C04270=1092.940,-90.083,-50.022,174.964,15.588,152.351
C04271=1092.934,-90.332,-50.011,174.962,15.588,152.351
C04272=1092.928,-90.582,-50.001,174.961,15.588,152.351
C04273=1092.922,-90.832,-49.990,174.959,15.586,152.351
C04274=1092.915,-91.082,-49.980,174.957,15.586,152.352
C04275=1092.910,-91.332,-49.970,174.955,15.585,152.352
C04276=1092.903,-91.581,-49.959,174.955,15.584,152.352
C04277=1092.898,-91.831,-49.949,174.953,15.584,152.352
C04278=1092.891,-92.080,-49.939,174.951,15.583,152.353
C04279=1092.886,-92.330,-49.929,174.949,15.582,152.353
C04280=1092.879,-92.579,-49.919,174.948,15.582,152.353
C04281=1092.874,-92.830,-49.908,174.946,15.581,152.353
C04282=1092.868,-93.079,-49.898,174.944,15.581,152.353
C04283=1092.862,-93.329,-49.888,174.943,15.580,152.354
C04284=1092.855,-93.579,-49.877,174.942,15.579,152.354
C04285=1092.850,-93.829,-49.867,174.940,15.579,152.354
C04286=1092.843,-94.078,-49.857,174.938,15.578,152.354
C04287=1092.838,-94.328,-49.847,174.936,15.577,152.355
C04288=1092.831,-94.577,-49.836,174.935,15.577,152.355
C04289=1092.826,-94.827,-49.826,174.933,15.576,152.355
C04290=1092.819,-95.077,-49.816,174.931,15.575,152.355
C04291=1092.814,-95.327,-49.806,174.930,15.575,152.355
C04292=1092.808,-95.576,-49.796,174.929,15.574,152.355
C04293=1092.802,-95.826,-49.785,174.927,15.574,152.356
C04294=1092.796,-96.076,-49.776,174.925,15.573,152.356
C04295=1092.790,-96.325,-49.765,174.923,15.572,152.356
C04296=1092.783,-96.600,-49.754,174.921,15.571,152.356
C04297=1092.776,-96.875,-49.742,174.920,15.571,152.357
C04298=1092.771,-97.150,-49.732,174.918,15.570,152.357
C04299=1092.763,-97.425,-49.720,174.917,15.570,152.357
C04300=1092.758,-97.675,-49.710,174.915,15.569,152.357
C04301=1092.751,-97.924,-49.700,174.913,15.568,152.358
C04302=1092.745,-98.174,-49.690,174.912,15.568,152.358
C04303=1092.740,-98.424,-49.680,174.910,15.567,152.358
C04304=1092.733,-98.673,-49.670,174.908,15.566,152.358
C04305=1092.727,-98.923,-49.660,174.906,15.566,152.359
C04306=1092.721,-99.174,-49.650,174.905,15.566,152.359
C04307=1092.715,-99.423,-49.640,174.903,15.565,152.359
C04308=1092.709,-99.673,-49.630,174.901,15.564,152.359
C04309=1092.702,-99.923,-49.620,174.901,15.564,152.359
C04310=1092.697,-100.172,-49.610,174.899,15.563,152.360
C04311=1092.690,-100.422,-49.600,174.897,15.562,152.360
C04312=1092.684,-100.672,-49.590,174.896,15.562,152.360
C04313=1092.679,-100.921,-49.580,174.894,15.562,152.360
C04314=1092.672,-101.171,-49.570,174.892,15.561,152.361
C04315=1092.666,-101.421,-49.560,174.890,15.560,152.361
C04316=1092.660,-101.670,-49.550,174.889,15.560,152.361
C04317=1092.654,-101.920,-49.540,174.887,15.559,152.361
C04318=1092.648,-102.170,-49.530,174.885,15.558,152.361
C04319=1092.642,-102.419,-49.520,174.884,15.558,152.362
C04320=1092.636,-102.669,-49.510,174.882,15.558,152.362
C04321=1092.630,-102.919,-49.500,174.880,15.557,152.362
C04322=1092.624,-103.169,-49.491,174.879,15.557,152.362
C04323=1092.617,-103.418,-49.481,174.877,15.556,152.363
C04324=1092.612,-103.668,-49.470,174.876,15.556,152.363
C04325=1092.606,-103.918,-49.461,174.875,15.555,152.363
C04326=1092.600,-104.168,-49.451,174.873,15.554,152.363
C04327=1092.593,-104.417,-49.441,174.871,15.554,152.364
C04328=1092.588,-104.667,-49.431,174.869,15.553,152.364
C04329=1092.581,-104.917,-49.421,174.868,15.553,152.364
C04330=1092.575,-105.167,-49.412,174.866,15.552,152.364
C04331=1092.569,-105.416,-49.402,174.864,15.552,152.365
C04332=1092.563,-105.666,-49.392,174.863,15.552,152.365
C04333=1092.557,-105.916,-49.382,174.861,15.551,152.365
C04334=1092.551,-106.165,-49.372,174.859,15.550,152.365
C04335=1092.545,-106.415,-49.362,174.858,15.550,152.366
C04336=1092.539,-106.665,-49.353,174.857,15.549,152.366
C04337=1092.532,-106.914,-49.343,174.855,15.548,152.366
C04338=1092.527,-107.164,-49.332,174.853,15.548,152.366
C04339=1092.521,-107.414,-49.323,174.852,15.548,152.366
C04340=1092.514,-107.664,-49.313,174.850,15.547,152.367
C04341=1092.508,-107.914,-49.304,174.849,15.547,152.367
C04342=1092.502,-108.164,-49.294,174.847,15.546,152.367
C04343=1092.496,-108.413,-49.284,174.845,15.545,152.367
C04344=1092.489,-108.663,-49.274,174.844,15.545,152.368
C04345=1092.484,-108.913,-49.264,174.842,15.545,152.368
C04346=1092.478,-109.162,-49.255,174.841,15.545,152.368
C04347=1092.472,-109.412,-49.245,174.839,15.544,152.368
C04348=1092.466,-109.662,-49.235,174.837,15.543,152.369
C04349=1092.459,-109.912,-49.226,174.836,15.543,152.369
C04350=1092.453,-110.162,-49.216,174.834,15.543,152.369
C04351=1092.447,-110.411,-49.207,174.832,15.542,152.369
C04352=1092.441,-110.661,-49.197,174.831,15.542,152.370
C04353=1092.434,-110.910,-49.187,174.829,15.541,152.370
C04354=1092.428,-111.160,-49.177,174.827,15.541,152.370
C04355=1092.422,-111.410,-49.168,174.826,15.540,152.370
C04356=1092.416,-111.659,-49.159,174.824,15.540,152.371
C04357=1092.410,-111.909,-49.149,174.822,15.539,152.371
C04358=1092.405,-112.159,-49.139,174.821,15.539,152.371
C04359=1092.399,-112.409,-49.129,174.819,15.538,152.371
C04360=1092.391,-112.676,-49.119,174.817,15.538,152.372
C04361=1092.385,-112.944,-49.109,174.816,15.538,152.372
C04362=1092.379,-113.211,-49.098,174.814,15.537,152.372
C04363=1092.372,-113.478,-49.088,174.812,15.536,152.373
C04364=1092.366,-113.727,-49.079,174.811,15.537,152.373
C04365=1092.359,-113.977,-49.069,174.809,15.536,152.373
C04366=1092.354,-114.226,-49.060,174.807,15.535,152.373
C04367=1092.348,-114.476,-49.050,174.806,15.535,152.374
C04368=1092.341,-114.726,-49.041,174.804,15.535,152.374
C04369=1092.335,-114.976,-49.031,174.802,15.534,152.374
C04370=1092.329,-115.226,-49.022,174.801,15.534,152.374
C04371=1092.323,-115.475,-49.012,174.799,15.533,152.375
C04372=1092.317,-115.725,-49.002,174.798,15.533,152.375
C04373=1092.311,-115.975,-48.993,174.796,15.533,152.375
C04374=1092.304,-116.225,-48.983,174.794,15.532,152.375
C04375=1092.298,-116.475,-48.974,174.793,15.532,152.376
C04376=1092.292,-116.724,-48.964,174.791,15.531,152.376
C04377=1092.286,-116.974,-48.955,174.790,15.531,152.376
C04378=1092.280,-117.223,-48.945,174.788,15.530,152.376
C04379=1092.274,-117.474,-48.937,174.786,15.530,152.377
C04380=1092.268,-117.723,-48.927,174.785,15.530,152.377
C04381=1092.262,-117.973,-48.917,174.783,15.530,152.377
C04382=1092.256,-118.223,-48.908,174.782,15.529,152.378
C04383=1092.250,-118.473,-48.898,174.780,15.529,152.378
C04384=1092.243,-118.722,-48.889,174.778,15.528,152.378
C04385=1092.237,-118.972,-48.880,174.777,15.528,152.378
C04386=1092.231,-119.222,-48.870,174.775,15.527,152.379
C04387=1092.225,-119.471,-48.861,174.774,15.527,152.379
C04388=1092.219,-119.721,-48.851,174.772,15.527,152.379
C04389=1092.213,-119.971,-48.842,174.770,15.526,152.380
C04390=1092.207,-120.221,-48.833,174.769,15.526,152.380
C04391=1092.201,-120.471,-48.823,174.767,15.526,152.380
C04392=1092.194,-120.721,-48.814,174.766,15.526,152.380
C04393=1092.188,-120.970,-48.805,174.764,15.525,152.381
C04394=1092.182,-121.219,-48.796,174.763,15.525,152.381
C04395=1092.176,-121.469,-48.786,174.761,15.525,152.381
C04396=1092.170,-121.719,-48.777,174.759,15.524,152.381
C04397=1092.164,-121.969,-48.768,174.758,15.524,152.382
C04398=1092.158,-122.219,-48.758,174.756,15.523,152.382
C04399=1092.151,-122.469,-48.749,174.755,15.523,152.382
C04400=1092.144,-122.718,-48.740,174.753,15.523,152.382
C04401=1092.139,-122.967,-48.730,174.751,15.522,152.383
C04402=1092.133,-123.218,-48.722,174.749,15.522,152.383
C04403=1092.127,-123.468,-48.712,174.747,15.522,152.383
C04404=1092.121,-123.717,-48.702,174.746,15.522,152.384
C04405=1092.115,-123.967,-48.693,174.744,15.521,152.384
C04406=1092.108,-124.217,-48.684,174.743,15.521,152.384
C04407=1092.102,-124.466,-48.675,174.741,15.521,152.384
C04408=1092.096,-124.716,-48.666,174.740,15.521,152.385
C04409=1092.090,-124.966,-48.656,174.738,15.520,152.385
C04410=1092.084,-125.216,-48.647,174.736,15.519,152.385
C04411=1092.077,-125.465,-48.638,174.735,15.519,152.385
C04412=1092.071,-125.716,-48.629,174.733,15.519,152.386
C04413=1092.065,-125.965,-48.620,174.732,15.519,152.386
C04414=1092.059,-126.215,-48.610,174.730,15.518,152.386
C04415=1092.052,-126.464,-48.601,174.729,15.518,152.387
C04416=1092.047,-126.715,-48.592,174.727,15.518,152.387
C04417=1092.040,-126.964,-48.583,174.726,15.518,152.387
C04418=1092.034,-127.213,-48.574,174.724,15.517,152.388
C04419=1092.028,-127.464,-48.565,174.722,15.517,152.388
C04420=1092.022,-127.723,-48.556,174.720,15.517,152.388
C04421=1092.016,-127.983,-48.546,174.718,15.517,152.388
C04422=1092.010,-128.242,-48.536,174.718,15.516,152.389
C04423=1092.015,-128.499,-48.524,174.717,15.513,152.388
C04424=1091.609,-128.520,-48.641,174.673,15.620,152.418
C04425=1091.604,-128.263,-48.653,174.674,15.624,152.418
C04426=1091.608,-128.004,-48.663,174.675,15.624,152.418
C04427=1091.615,-127.744,-48.673,174.677,15.625,152.418
C04428=1091.620,-127.485,-48.682,174.679,15.625,152.418
C04429=1091.627,-127.236,-48.692,174.680,15.625,152.417
C04430=1091.634,-126.986,-48.701,174.682,15.626,152.417
C04431=1091.639,-126.736,-48.710,174.683,15.626,152.417
C04432=1091.646,-126.486,-48.719,174.685,15.627,152.417
C04433=1091.652,-126.237,-48.728,174.686,15.626,152.416
C04434=1091.658,-125.987,-48.737,174.688,15.627,152.416
C04435=1091.664,-125.737,-48.746,174.689,15.627,152.416
C04436=1091.670,-125.487,-48.756,174.691,15.627,152.415
C04437=1091.677,-125.238,-48.765,174.693,15.628,152.415
C04438=1091.683,-124.988,-48.774,174.694,15.628,152.415
C04439=1091.689,-124.738,-48.784,174.697,15.628,152.414
C04440=1091.695,-124.488,-48.792,174.698,15.628,152.414
C04441=1091.701,-124.239,-48.802,174.700,15.629,152.414
C04442=1091.708,-123.989,-48.811,174.701,15.629,152.414
C04443=1091.714,-123.739,-48.820,174.703,15.630,152.413
C04444=1091.720,-123.489,-48.829,174.704,15.630,152.413
C04445=1091.725,-123.240,-48.839,174.706,15.630,152.413
C04446=1091.732,-122.990,-48.848,174.708,15.631,152.413
C04447=1091.738,-122.740,-48.858,174.709,15.631,152.412
C04448=1091.745,-122.491,-48.867,174.711,15.631,152.412
C04449=1091.750,-122.240,-48.875,174.712,15.631,152.412
C04450=1091.757,-121.990,-48.885,174.714,15.632,152.412
C04451=1091.763,-121.741,-48.895,174.716,15.633,152.411
C04452=1091.768,-121.492,-48.904,174.717,15.633,152.411
C04453=1091.775,-121.242,-48.913,174.719,15.633,152.411
C04454=1091.781,-120.992,-48.922,174.720,15.633,152.410
C04455=1091.788,-120.743,-48.932,174.722,15.634,152.410
C04456=1091.793,-120.492,-48.941,174.724,15.634,152.410
C04457=1091.800,-120.242,-48.950,174.725,15.634,152.410
C04458=1091.806,-119.992,-48.960,174.727,15.635,152.409
C04459=1091.811,-119.743,-48.969,174.728,15.635,152.409
C04460=1091.818,-119.494,-48.979,174.730,15.636,152.409
C04461=1091.824,-119.244,-48.988,174.732,15.636,152.409
C04462=1091.830,-118.994,-48.998,174.733,15.637,152.408
C04463=1091.837,-118.745,-49.007,174.735,15.637,152.408
C04464=1091.843,-118.494,-49.016,174.736,15.637,152.408
C04465=1091.849,-118.244,-49.025,174.738,15.638,152.408
C04466=1091.855,-117.995,-49.035,174.740,15.639,152.407
C04467=1091.861,-117.745,-49.044,174.741,15.638,152.407
C04468=1091.867,-117.496,-49.054,174.743,15.639,152.407
C04469=1091.873,-117.246,-49.063,174.744,15.639,152.407
C04470=1091.879,-116.996,-49.073,174.746,15.639,152.406
C04471=1091.885,-116.746,-49.082,174.748,15.640,152.406
C04472=1091.891,-116.496,-49.092,174.749,15.640,152.406
C04473=1091.898,-116.247,-49.101,174.751,15.641,152.406
C04474=1091.904,-115.997,-49.111,174.752,15.641,152.405
C04475=1091.910,-115.747,-49.121,174.754,15.642,152.405
C04476=1091.916,-115.497,-49.130,174.756,15.642,152.405
C04477=1091.922,-115.248,-49.139,174.757,15.642,152.405
C04478=1091.928,-114.998,-49.149,174.759,15.643,152.404
C04479=1091.934,-114.749,-49.158,174.761,15.644,152.404
C04480=1091.940,-114.499,-49.168,174.762,15.644,152.404
C04481=1091.946,-114.249,-49.178,174.764,15.644,152.403
C04482=1091.953,-113.999,-49.187,174.765,15.644,152.403
C04483=1091.959,-113.749,-49.197,174.767,15.645,152.403
C04484=1091.965,-113.500,-49.206,174.769,15.646,152.403
C04485=1091.972,-113.232,-49.216,174.770,15.646,152.403
C04486=1091.978,-112.965,-49.226,174.772,15.646,152.402
C04487=1091.984,-112.697,-49.236,174.774,15.647,152.402
C04488=1091.991,-112.430,-49.247,174.776,15.648,152.402
C04489=1091.997,-112.180,-49.257,174.777,15.648,152.401
C04490=1092.003,-111.930,-49.266,174.779,15.649,152.401
C04491=1092.009,-111.680,-49.276,174.780,15.649,152.401
C04492=1092.016,-111.431,-49.285,174.782,15.649,152.401
C04493=1092.022,-111.181,-49.295,174.783,15.650,152.400
C04494=1092.028,-110.931,-49.305,174.785,15.651,152.400
C04495=1092.034,-110.681,-49.314,174.786,15.651,152.400
C04496=1092.040,-110.431,-49.324,174.788,15.651,152.400
C04497=1092.046,-110.182,-49.333,174.790,15.652,152.399
C04498=1092.053,-109.932,-49.343,174.791,15.652,152.399
C04499=1092.058,-109.682,-49.354,174.793,15.653,152.399
C04500=1092.064,-109.432,-49.363,174.795,15.653,152.399
C04501=1092.071,-109.183,-49.373,174.796,15.654,152.399
C04502=1092.077,-108.933,-49.382,174.798,15.655,152.398
C04503=1092.083,-108.683,-49.392,174.799,15.655,152.398
C04504=1092.089,-108.433,-49.402,174.801,15.655,152.398
C04505=1092.095,-108.183,-49.411,174.803,15.656,152.398
C04506=1092.102,-107.934,-49.421,174.804,15.656,152.397
C04507=1092.108,-107.684,-49.431,174.806,15.657,152.397
C04508=1092.113,-107.434,-49.441,174.808,15.657,152.397
C04509=1092.120,-107.185,-49.451,174.809,15.657,152.397
C04510=1092.126,-106.935,-49.460,174.811,15.658,152.396
C04511=1092.132,-106.685,-49.470,174.813,15.659,152.396
C04512=1092.138,-106.435,-49.479,174.814,15.660,152.396
C04513=1092.145,-106.186,-49.490,174.815,15.660,152.396
C04514=1092.150,-105.936,-49.500,174.817,15.661,152.395
C04515=1092.156,-105.687,-49.509,174.819,15.661,152.395
C04516=1092.162,-105.437,-49.519,174.820,15.661,152.395
C04517=1092.168,-105.187,-49.528,174.822,15.662,152.395
C04518=1092.174,-104.938,-49.539,174.824,15.663,152.394
C04519=1092.180,-104.688,-49.549,174.825,15.663,152.394
C04520=1092.186,-104.438,-49.558,174.827,15.664,152.394
C04521=1092.192,-104.188,-49.568,174.829,15.665,152.394
C04522=1092.199,-103.939,-49.578,174.830,15.665,152.394
C04523=1092.204,-103.689,-49.588,174.832,15.665,152.393
C04524=1092.210,-103.439,-49.598,174.834,15.666,152.393
C04525=1092.216,-103.189,-49.607,174.835,15.666,152.393
C04526=1092.223,-102.940,-49.618,174.836,15.667,152.393
C04527=1092.228,-102.690,-49.628,174.838,15.668,152.393
C04528=1092.235,-102.440,-49.638,174.840,15.668,152.392
C04529=1092.241,-102.190,-49.647,174.841,15.669,152.392
C04530=1092.247,-101.940,-49.658,174.843,15.669,152.392
C04531=1092.253,-101.691,-49.668,174.845,15.670,152.391
C04532=1092.259,-101.441,-49.677,174.846,15.670,152.391
C04533=1092.266,-101.192,-49.688,174.848,15.671,152.391
C04534=1092.271,-100.941,-49.698,174.850,15.672,152.391
C04535=1092.277,-100.692,-49.707,174.851,15.672,152.391
C04536=1092.284,-100.443,-49.718,174.853,15.673,152.390
C04537=1092.290,-100.193,-49.727,174.854,15.674,152.390
C04538=1092.296,-99.943,-49.737,174.856,15.674,152.390
C04539=1092.302,-99.693,-49.748,174.857,15.674,152.390
C04540=1092.308,-99.444,-49.757,174.859,15.675,152.390
C04541=1092.314,-99.194,-49.767,174.861,15.676,152.389
C04542=1092.320,-98.944,-49.778,174.862,15.676,152.389
C04543=1092.326,-98.695,-49.787,174.864,15.677,152.389
C04544=1092.332,-98.444,-49.797,174.866,15.678,152.389
C04545=1092.338,-98.195,-49.808,174.867,15.678,152.388
C04546=1092.344,-97.945,-49.817,174.869,15.678,152.388
C04547=1092.350,-97.695,-49.828,174.870,15.679,152.388
C04548=1092.357,-97.445,-49.838,174.872,15.680,152.388
C04549=1092.363,-97.171,-49.849,174.874,15.681,152.388
C04550=1092.370,-96.896,-49.860,174.876,15.681,152.387
C04551=1092.376,-96.620,-49.871,174.878,15.682,152.387
C04552=1092.382,-96.345,-49.882,174.879,15.683,152.387
C04553=1092.389,-96.096,-49.893,174.880,15.683,152.387
C04554=1092.394,-95.846,-49.903,174.882,15.684,152.386
C04555=1092.401,-95.596,-49.913,174.884,15.685,152.386
C04556=1092.406,-95.346,-49.923,174.885,15.685,152.386
C04557=1092.413,-95.097,-49.934,174.887,15.686,152.386
C04558=1092.419,-94.847,-49.943,174.889,15.687,152.386
C04559=1092.424,-94.597,-49.953,174.890,15.688,152.385
C04560=1092.431,-94.348,-49.964,174.892,15.688,152.385
C04561=1092.436,-94.098,-49.974,174.893,15.689,152.385
C04562=1092.443,-93.849,-49.984,174.895,15.690,152.385
C04563=1092.449,-93.598,-49.995,174.897,15.690,152.385
C04564=1092.455,-93.349,-50.005,174.898,15.690,152.384
C04565=1092.461,-93.099,-50.015,174.900,15.692,152.384
C04566=1092.466,-92.849,-50.026,174.902,15.692,152.384
C04567=1092.473,-92.599,-50.035,174.903,15.693,152.384
C04568=1092.478,-92.350,-50.046,174.904,15.693,152.384
C04569=1092.485,-92.100,-50.056,174.906,15.694,152.383
C04570=1092.490,-91.851,-50.067,174.908,15.695,152.383
C04571=1092.496,-91.601,-50.076,174.910,15.696,152.383
C04572=1092.502,-91.351,-50.087,174.912,15.697,152.383
C04573=1092.508,-91.101,-50.097,174.913,15.697,152.383
C04574=1092.515,-90.851,-50.108,174.915,15.697,152.382
C04575=1092.521,-90.602,-50.118,174.916,15.698,152.382
C04576=1092.527,-90.352,-50.128,174.918,15.699,152.382
C04577=1092.533,-90.103,-50.139,174.919,15.699,152.382
C04578=1092.539,-89.853,-50.149,174.921,15.700,152.382
C04579=1092.545,-89.604,-50.159,174.923,15.701,152.381
C04580=1092.550,-89.353,-50.169,174.924,15.702,152.381
C04581=1092.557,-89.103,-50.181,174.925,15.702,152.381
C04582=1092.563,-88.854,-50.191,174.927,15.703,152.381
C04583=1092.569,-88.604,-50.201,174.929,15.704,152.381
C04584=1092.575,-88.355,-50.211,174.931,15.705,152.380
C04585=1092.581,-88.105,-50.222,174.933,15.705,152.380
C04586=1092.587,-87.855,-50.232,174.933,15.706,152.380
C04587=1092.593,-87.606,-50.243,174.935,15.707,152.380
C04588=1092.599,-87.355,-50.253,174.937,15.707,152.379
C04589=1092.605,-87.106,-50.263,174.939,15.708,152.379
C04590=1092.611,-86.856,-50.274,174.941,15.709,152.379
C04591=1092.617,-86.607,-50.284,174.942,15.709,152.379
C04592=1092.623,-86.357,-50.295,174.943,15.710,152.379
C04593=1092.630,-86.107,-50.305,174.945,15.711,152.379
C04594=1092.635,-85.857,-50.316,174.947,15.712,152.378
C04595=1092.641,-85.608,-50.326,174.949,15.713,152.378
C04596=1092.648,-85.359,-50.337,174.950,15.713,152.378
C04597=1092.653,-85.108,-50.347,174.952,15.714,152.378
C04598=1092.660,-84.859,-50.358,174.953,15.715,152.378
C04599=1092.666,-84.609,-50.368,174.955,15.715,152.377
C04600=1092.671,-84.359,-50.379,174.957,15.717,152.377
C04601=1092.678,-84.110,-50.389,174.958,15.717,152.377
C04602=1092.684,-83.860,-50.400,174.960,15.717,152.377
C04603=1092.690,-83.610,-50.411,174.962,15.719,152.377
C04604=1092.696,-83.360,-50.421,174.963,15.719,152.376
C04605=1092.702,-83.111,-50.431,174.965,15.720,152.376
C04606=1092.708,-82.862,-50.442,174.966,15.720,152.376
C04607=1092.715,-82.611,-50.453,174.968,15.721,152.376
C04608=1092.720,-82.361,-50.463,174.970,15.722,152.376
C04609=1092.727,-82.112,-50.473,174.972,15.723,152.375
C04610=1092.732,-81.863,-50.484,174.973,15.724,152.375
C04611=1092.739,-81.612,-50.496,174.974,15.724,152.375
C04612=1092.745,-81.363,-50.505,174.976,15.725,152.375
C04613=1092.752,-81.091,-50.517,174.978,15.725,152.375
C04614=1092.758,-80.817,-50.529,174.980,15.727,152.374
C04615=1092.764,-80.545,-50.541,174.982,15.727,152.374
C04616=1092.771,-80.271,-50.552,174.983,15.728,152.374
C04617=1092.778,-80.022,-50.563,174.985,15.729,152.374
C04618=1092.784,-79.773,-50.573,174.987,15.730,152.374
C04619=1092.789,-79.523,-50.584,174.989,15.731,152.373
C04620=1092.795,-79.272,-50.595,174.990,15.732,152.373
C04621=1092.801,-79.023,-50.606,174.991,15.732,152.373
C04622=1092.808,-78.774,-50.616,174.993,15.733,152.373
C04623=1092.813,-78.524,-50.627,174.995,15.734,152.373
C04624=1092.820,-78.274,-50.638,174.997,15.735,152.372
C04625=1092.825,-78.024,-50.649,174.998,15.736,152.372
C04626=1092.831,-77.775,-50.660,175.000,15.736,152.372
C04627=1092.837,-77.525,-50.670,175.001,15.737,152.372
C04628=1092.844,-77.275,-50.681,175.003,15.738,152.372
C04629=1092.849,-77.025,-50.692,175.004,15.739,152.372
C04630=1092.855,-76.776,-50.702,175.006,15.740,152.371
C04631=1092.861,-76.526,-50.713,175.008,15.741,152.371
C04632=1092.867,-76.276,-50.725,175.010,15.741,152.371
C04633=1092.873,-76.027,-50.735,175.012,15.742,152.371
C04634=1092.879,-75.778,-50.746,175.013,15.743,152.371
C04635=1092.885,-75.528,-50.757,175.014,15.743,152.370
C04636=1092.892,-75.278,-50.768,175.016,15.744,152.370
C04637=1092.897,-75.028,-50.779,175.018,15.745,152.370
C04638=1092.903,-74.779,-50.790,175.020,15.746,152.370
C04639=1092.909,-74.528,-50.800,175.021,15.747,152.370
C04640=1092.915,-74.279,-50.811,175.023,15.748,152.370
C04641=1092.920,-74.029,-50.822,175.024,15.748,152.369
C04642=1092.926,-73.780,-50.833,175.026,15.749,152.369
C04643=1092.933,-73.529,-50.844,175.027,15.751,152.369
C04644=1092.938,-73.280,-50.855,175.029,15.751,152.369
C04645=1092.944,-73.031,-50.866,175.031,15.752,152.369
C04646=1092.950,-72.781,-50.877,175.033,15.753,152.369
C04647=1092.956,-72.531,-50.888,175.034,15.754,152.368
C04648=1092.962,-72.281,-50.899,175.036,15.755,152.368
C04649=1092.968,-72.032,-50.910,175.038,15.756,152.368
C04650=1092.973,-71.782,-50.920,175.039,15.757,152.368
C04651=1092.980,-71.532,-50.932,175.040,15.757,152.368
C04652=1092.985,-71.283,-50.943,175.042,15.758,152.368
C04653=1092.991,-71.033,-50.953,175.044,15.759,152.367
C04654=1092.998,-70.783,-50.965,175.046,15.760,152.367
C04655=1093.003,-70.533,-50.976,175.047,15.761,152.367
C04656=1093.009,-70.284,-50.986,175.049,15.762,152.367
C04657=1093.015,-70.035,-50.997,175.051,15.763,152.367
C04658=1093.021,-69.785,-51.009,175.053,15.764,152.367
C04659=1093.027,-69.535,-51.020,175.053,15.764,152.366
C04660=1093.033,-69.286,-51.031,175.055,15.765,152.366
C04661=1093.038,-69.035,-51.043,175.057,15.766,152.366
C04662=1093.044,-68.786,-51.054,175.058,15.767,152.366
C04663=1093.050,-68.536,-51.065,175.060,15.768,152.366
C04664=1093.056,-68.286,-51.076,175.062,15.769,152.366
C04665=1093.062,-68.037,-51.087,175.064,15.770,152.365
C04666=1093.068,-67.787,-51.098,175.065,15.771,152.365
C04667=1093.074,-67.537,-51.109,175.067,15.772,152.365
C04668=1093.080,-67.288,-51.120,175.069,15.773,152.365
C04669=1093.086,-67.039,-51.131,175.070,15.774,152.365
C04670=1093.092,-66.789,-51.143,175.072,15.774,152.365
C04671=1093.097,-66.539,-51.154,175.073,15.775,152.364
C04672=1093.103,-66.289,-51.165,175.075,15.776,152.364
C04673=1093.109,-66.039,-51.176,175.077,15.777,152.364
C04674=1093.115,-65.790,-51.187,175.078,15.778,152.364
C04675=1093.121,-65.541,-51.199,175.080,15.779,152.364
C04676=1093.127,-65.291,-51.210,175.082,15.780,152.364
C04677=1093.134,-65.020,-51.222,175.083,15.781,152.364
C04678=1093.140,-64.749,-51.234,175.085,15.782,152.363
C04679=1093.146,-64.479,-51.246,175.087,15.783,152.363
C04680=1093.152,-64.208,-51.258,175.089,15.784,152.363
C04681=1093.159,-63.958,-51.269,175.090,15.785,152.363
C04682=1093.165,-63.709,-51.281,175.092,15.786,152.363
C04683=1093.171,-63.459,-51.292,175.094,15.787,152.362
C04684=1093.177,-63.209,-51.303,175.096,15.788,152.362
C04685=1093.182,-62.960,-51.315,175.097,15.789,152.362
C04686=1093.188,-62.710,-51.327,175.099,15.790,152.362
C04687=1093.194,-62.461,-51.337,175.101,15.790,152.362
C04688=1093.201,-62.210,-51.349,175.102,15.792,152.362
C04689=1093.206,-61.961,-51.360,175.104,15.793,152.361
C04690=1093.212,-61.712,-51.371,175.105,15.793,152.361
C04691=1093.218,-61.462,-51.383,175.107,15.794,152.361
C04692=1093.224,-61.212,-51.394,175.108,15.795,152.361
C04693=1093.230,-60.962,-51.406,175.110,15.796,152.361
C04694=1093.236,-60.713,-51.417,175.112,15.797,152.361
C04695=1093.242,-60.463,-51.428,175.114,15.798,152.360
C04696=1093.248,-60.214,-51.440,175.115,15.799,152.360
C04697=1093.254,-59.963,-51.451,175.117,15.800,152.360
C04698=1093.260,-59.714,-51.462,175.119,15.801,152.360
C04699=1093.266,-59.464,-51.474,175.120,15.802,152.360
C04700=1093.272,-59.215,-51.485,175.122,15.802,152.360
C04701=1093.277,-58.965,-51.497,175.124,15.804,152.359
C04702=1093.284,-58.715,-51.508,175.126,15.805,152.359
C04703=1093.290,-58.466,-51.519,175.127,15.805,152.359
C04704=1093.296,-58.216,-51.531,175.129,15.807,152.359
C04705=1093.302,-57.967,-51.542,175.131,15.807,152.359
C04706=1093.308,-57.716,-51.554,175.133,15.808,152.359
C04707=1093.313,-57.467,-51.565,175.134,15.810,152.359
C04708=1093.320,-57.217,-51.577,175.136,15.810,152.358
C04709=1093.326,-56.968,-51.588,175.137,15.811,152.358
C04710=1093.332,-56.718,-51.600,175.138,15.812,152.358
C04711=1093.337,-56.468,-51.611,175.140,15.813,152.358
C04712=1093.344,-56.219,-51.623,175.142,15.814,152.358
C04713=1093.350,-55.969,-51.634,175.144,15.815,152.357
C04714=1093.356,-55.719,-51.645,175.145,15.816,152.357
C04715=1093.361,-55.470,-51.657,175.147,15.817,152.357
C04716=1093.368,-55.220,-51.669,175.149,15.818,152.357
C04717=1093.374,-54.970,-51.681,175.151,15.819,152.357
C04718=1093.380,-54.721,-51.692,175.152,15.819,152.357
C04719=1093.386,-54.471,-51.704,175.154,15.821,152.357
C04720=1093.392,-54.221,-51.715,175.156,15.822,152.356
C04721=1093.398,-53.972,-51.727,175.158,15.822,152.356
C04722=1093.403,-53.722,-51.738,175.159,15.824,152.356
C04723=1093.410,-53.472,-51.750,175.161,15.824,152.356
C04724=1093.416,-53.223,-51.761,175.163,15.825,152.356
C04725=1093.422,-52.973,-51.773,175.164,15.827,152.356
C04726=1093.428,-52.723,-51.785,175.166,15.827,152.355
C04727=1093.434,-52.474,-51.797,175.168,15.828,152.355
C04728=1093.440,-52.224,-51.808,175.169,15.830,152.355
C04729=1093.446,-51.975,-51.820,175.171,15.830,152.355
C04730=1093.452,-51.724,-51.831,175.173,15.831,152.355
C04731=1093.458,-51.476,-51.843,175.175,15.832,152.355
C04732=1093.465,-51.226,-51.855,175.176,15.833,152.354
C04733=1093.470,-50.976,-51.867,175.178,15.834,152.354
C04734=1093.476,-50.727,-51.878,175.180,15.835,152.354
C04735=1093.483,-50.476,-51.890,175.181,15.836,152.354
C04736=1093.488,-50.227,-51.902,175.183,15.837,152.354
C04737=1093.494,-49.977,-51.913,175.185,15.838,152.354
C04738=1093.500,-49.728,-51.925,175.186,15.839,152.353
C04739=1093.506,-49.478,-51.937,175.188,15.840,152.353
C04740=1093.511,-49.229,-51.949,175.190,15.841,152.353
C04741=1093.518,-48.959,-51.962,175.192,15.842,152.353
C04742=1093.524,-48.689,-51.974,175.193,15.843,152.353
C04743=1093.530,-48.420,-51.987,175.195,15.844,152.353
C04744=1093.537,-48.151,-52.000,175.197,15.845,152.353
C04745=1093.543,-47.901,-52.012,175.198,15.846,152.352
C04746=1093.549,-47.652,-52.024,175.200,15.847,152.352
C04747=1093.555,-47.402,-52.036,175.202,15.848,152.352
C04748=1093.560,-47.153,-52.047,175.203,15.849,152.352
C04749=1093.566,-46.903,-52.060,175.206,15.851,152.352
C04750=1093.572,-46.654,-52.071,175.207,15.852,152.352
C04751=1093.578,-46.403,-52.083,175.209,15.853,152.351
C04752=1093.584,-46.154,-52.095,175.211,15.854,152.351
C04753=1093.590,-45.905,-52.107,175.212,15.855,152.351
C04754=1093.596,-45.654,-52.119,175.214,15.856,152.351
C04755=1093.601,-45.405,-52.131,175.216,15.857,152.351
C04756=1093.608,-45.156,-52.143,175.217,15.858,152.351
C04757=1093.614,-44.905,-52.155,175.219,15.859,152.351
C04758=1093.619,-44.656,-52.167,175.221,15.860,152.350
C04759=1093.626,-44.406,-52.179,175.223,15.861,152.350
C04760=1093.631,-44.157,-52.191,175.224,15.862,152.350
C04761=1093.637,-43.907,-52.202,175.226,15.863,152.350
C04762=1093.643,-43.657,-52.215,175.228,15.864,152.350
C04763=1093.648,-43.408,-52.227,175.229,15.865,152.350
C04764=1093.655,-43.158,-52.239,175.231,15.867,152.350
C04765=1093.661,-42.908,-52.251,175.233,15.867,152.349
C04766=1093.667,-42.659,-52.262,175.234,15.868,152.349
C04767=1093.673,-42.409,-52.275,175.236,15.870,152.349
C04768=1093.678,-42.160,-52.287,175.238,15.870,152.349
C04769=1093.685,-41.910,-52.299,175.239,15.871,152.349
C04770=1093.690,-41.660,-52.311,175.241,15.873,152.349
C04771=1093.695,-41.411,-52.323,175.243,15.874,152.349
C04772=1093.702,-41.161,-52.335,175.245,15.874,152.348
C04773=1093.708,-40.911,-52.348,175.246,15.876,152.348
C04774=1093.714,-40.662,-52.359,175.248,15.877,152.348
C04775=1093.720,-40.412,-52.372,175.250,15.877,152.348
C04776=1093.726,-40.162,-52.383,175.251,15.879,152.348
C04777=1093.732,-39.913,-52.395,175.253,15.880,152.348
C04778=1093.738,-39.663,-52.408,175.255,15.880,152.347
C04779=1093.743,-39.413,-52.420,175.256,15.882,152.347
C04780=1093.750,-39.164,-52.432,175.259,15.883,152.347
C04781=1093.755,-38.915,-52.444,175.260,15.884,152.347
C04782=1093.761,-38.665,-52.457,175.262,15.885,152.347
C04783=1093.768,-38.415,-52.469,175.264,15.886,152.347
C04784=1093.773,-38.166,-52.481,175.265,15.887,152.347
C04785=1093.779,-37.915,-52.493,175.267,15.889,152.347
C04786=1093.785,-37.666,-52.505,175.269,15.889,152.346
C04787=1093.790,-37.416,-52.518,175.270,15.890,152.346
C04788=1093.797,-37.167,-52.530,175.272,15.892,152.346
C04789=1093.803,-36.917,-52.542,175.274,15.893,152.346
C04790=1093.808,-36.668,-52.554,175.276,15.893,152.346
C04791=1093.814,-36.418,-52.567,175.277,15.895,152.346
C04792=1093.820,-36.168,-52.579,175.279,15.896,152.346
C04793=1093.825,-35.919,-52.592,175.280,15.897,152.345
C04794=1093.832,-35.669,-52.604,175.282,15.898,152.345
C04795=1093.838,-35.419,-52.616,175.284,15.899,152.345
C04796=1093.843,-35.170,-52.628,175.286,15.901,152.345
C04797=1093.849,-34.920,-52.641,175.288,15.902,152.345
C04798=1093.855,-34.670,-52.653,175.290,15.902,152.345
C04799=1093.860,-34.421,-52.666,175.291,15.904,152.344
C04800=1093.867,-34.172,-52.678,175.293,15.905,152.344
C04801=1093.873,-33.922,-52.690,175.295,15.906,152.344
C04802=1093.879,-33.672,-52.703,175.296,15.907,152.344
C04803=1093.884,-33.423,-52.715,175.298,15.908,152.344
C04804=1093.890,-33.173,-52.727,175.300,15.909,152.344
C04805=1093.896,-32.904,-52.741,175.301,15.910,152.344
C04806=1093.903,-32.636,-52.754,175.304,15.911,152.343
C04807=1093.909,-32.366,-52.767,175.305,15.912,152.343
C04808=1093.915,-32.097,-52.781,175.307,15.914,152.343
C04809=1093.921,-31.847,-52.793,175.309,15.915,152.343
C04810=1093.927,-31.598,-52.805,175.311,15.915,152.343
C04811=1093.933,-31.348,-52.818,175.312,15.917,152.343
C04812=1093.939,-31.098,-52.830,175.314,15.918,152.343
C04813=1093.945,-30.849,-52.843,175.316,15.920,152.342
C04814=1093.951,-30.600,-52.856,175.318,15.920,152.342
C04815=1093.956,-30.350,-52.868,175.320,15.921,152.342
C04816=1093.962,-30.100,-52.881,175.321,15.923,152.342
C04817=1093.968,-29.850,-52.894,175.323,15.923,152.342
C04818=1093.974,-29.601,-52.906,175.325,15.924,152.342
C04819=1093.980,-29.351,-52.918,175.326,15.926,152.342
C04820=1093.986,-29.102,-52.931,175.328,15.927,152.341
C04821=1093.992,-28.852,-52.944,175.330,15.927,152.341
C04822=1093.998,-28.602,-52.956,175.331,15.929,152.341
C04823=1094.004,-28.353,-52.968,175.334,15.930,152.341
C04824=1094.009,-28.103,-52.981,175.335,15.931,152.341
C04825=1094.015,-27.853,-52.993,175.337,15.932,152.341
C04826=1094.022,-27.604,-53.007,175.339,15.933,152.340
C04827=1094.027,-27.354,-53.019,175.341,15.934,152.340
C04828=1094.033,-27.104,-53.032,175.342,15.935,152.340
C04829=1094.039,-26.855,-53.044,175.344,15.936,152.340
C04830=1094.045,-26.606,-53.057,175.346,15.937,152.340
C04831=1094.051,-26.356,-53.070,175.347,15.939,152.340
C04832=1094.057,-26.106,-53.082,175.349,15.940,152.340
C04833=1094.062,-25.857,-53.095,175.351,15.941,152.339
C04834=1094.068,-25.608,-53.108,175.353,15.942,152.339
C04835=1094.074,-25.358,-53.120,175.355,15.943,152.339
C04836=1094.080,-25.108,-53.133,175.356,15.944,152.339
C04837=1094.085,-24.858,-53.146,175.358,15.945,152.339
C04838=1094.091,-24.609,-53.159,175.360,15.946,152.339
C04839=1094.097,-24.359,-53.172,175.361,15.947,152.339
C04840=1094.103,-24.109,-53.184,175.363,15.949,152.339
C04841=1094.109,-23.859,-53.197,175.365,15.950,152.338
C04842=1094.115,-23.610,-53.210,175.367,15.951,152.338
C04843=1094.121,-23.360,-53.222,175.369,15.952,152.338
C04844=1094.126,-23.111,-53.235,175.370,15.953,152.338
C04845=1094.131,-22.861,-53.249,175.372,15.955,152.338
C04846=1094.137,-22.612,-53.261,175.374,15.955,152.338
C04847=1094.143,-22.362,-53.274,175.376,15.956,152.338
C04848=1094.149,-22.112,-53.287,175.377,15.958,152.337
C04849=1094.155,-21.863,-53.299,175.380,15.959,152.337
C04850=1094.162,-21.613,-53.313,175.381,15.960,152.337
C04851=1094.167,-21.364,-53.325,175.383,15.961,152.337
C04852=1094.172,-21.114,-53.338,175.385,15.962,152.337
C04853=1094.178,-20.865,-53.351,175.386,15.963,152.337
C04854=1094.184,-20.615,-53.364,175.388,15.964,152.336
C04855=1094.190,-20.365,-53.377,175.390,15.965,152.336
C04856=1094.196,-20.116,-53.390,175.392,15.967,152.336
C04857=1094.202,-19.866,-53.402,175.394,15.968,152.336
C04858=1094.208,-19.616,-53.416,175.396,15.969,152.336
C04859=1094.214,-19.366,-53.429,175.397,15.970,152.336
C04860=1094.219,-19.118,-53.442,175.399,15.971,152.336
C04861=1094.225,-18.868,-53.454,175.400,15.972,152.336
C04862=1094.231,-18.619,-53.467,175.402,15.973,152.335
C04863=1094.237,-18.369,-53.480,175.405,15.975,152.335
C04864=1094.243,-18.119,-53.494,175.406,15.976,152.335
C04865=1094.249,-17.869,-53.506,175.408,15.977,152.335
C04866=1094.255,-17.619,-53.519,175.410,15.978,152.335
C04867=1094.261,-17.370,-53.532,175.411,15.979,152.335
C04868=1094.267,-17.120,-53.545,175.413,15.980,152.335
C04869=1094.273,-16.851,-53.559,175.416,15.981,152.334
C04870=1094.279,-16.581,-53.573,175.417,15.983,152.334
C04871=1094.286,-16.311,-53.588,175.419,15.984,152.334
C04872=1094.292,-16.041,-53.602,175.422,15.985,152.334
C04873=1094.298,-15.792,-53.615,175.423,15.986,152.334
C04874=1094.304,-15.542,-53.628,175.425,15.987,152.334
C04875=1094.309,-15.292,-53.641,175.426,15.989,152.333
C04876=1094.316,-15.043,-53.654,175.428,15.989,152.333
C04877=1094.321,-14.793,-53.667,175.430,15.990,152.333
C04878=1094.327,-14.543,-53.681,175.432,15.992,152.333
C04879=1094.332,-14.294,-53.693,175.434,15.993,152.333
C04880=1094.338,-14.045,-53.706,175.436,15.994,152.333
C04881=1094.344,-13.795,-53.720,175.437,15.995,152.332
C04882=1094.350,-13.546,-53.733,175.439,15.996,152.332
C04883=1094.355,-13.296,-53.747,175.440,15.997,152.332
C04884=1094.361,-13.046,-53.759,175.443,15.999,152.332
C04885=1094.367,-12.797,-53.772,175.445,16.000,152.332
C04886=1094.373,-12.547,-53.786,175.446,16.001,152.332
C04887=1094.379,-12.297,-53.799,175.448,16.002,152.332
C04888=1094.384,-12.048,-53.813,175.450,16.003,152.331
C04889=1094.390,-11.798,-53.826,175.451,16.004,152.331
C04890=1094.396,-11.549,-53.838,175.454,16.006,152.331
C04891=1094.402,-11.299,-53.852,175.455,16.007,152.331
C04892=1094.408,-11.050,-53.866,175.457,16.008,152.331
C04893=1094.413,-10.800,-53.879,175.459,16.009,152.331
C04894=1094.419,-10.550,-53.892,175.461,16.010,152.331
C04895=1094.426,-10.301,-53.905,175.462,16.011,152.331
C04896=1094.431,-10.051,-53.918,175.465,16.012,152.330
C04897=1094.437,-9.802,-53.932,175.466,16.014,152.330
C04898=1094.443,-9.552,-53.946,175.468,16.015,152.330
C04899=1094.449,-9.303,-53.959,175.470,16.016,152.330
C04900=1094.454,-9.053,-53.972,175.472,16.017,152.330
C04901=1094.460,-8.803,-53.985,175.474,16.018,152.330
C04902=1094.466,-8.554,-53.999,175.476,16.019,152.329
C04903=1094.472,-8.304,-54.012,175.477,16.020,152.329
C04904=1094.478,-8.055,-54.025,175.479,16.021,152.329
C04905=1094.483,-7.805,-54.039,175.481,16.022,152.329
C04906=1094.489,-7.556,-54.052,175.483,16.024,152.329
C04907=1094.495,-7.306,-54.066,175.485,16.025,152.329
C04908=1094.501,-7.056,-54.079,175.486,16.026,152.329
C04909=1094.506,-6.807,-54.092,175.488,16.027,152.328
C04910=1094.513,-6.557,-54.106,175.490,16.028,152.328
C04911=1094.518,-6.308,-54.120,175.492,16.029,152.328
C04912=1094.524,-6.059,-54.133,175.494,16.031,152.328
C04913=1094.530,-5.808,-54.147,175.496,16.031,152.328
C04914=1094.536,-5.558,-54.160,175.497,16.033,152.328
C04915=1094.542,-5.309,-54.173,175.499,16.034,152.327
C04916=1094.548,-5.060,-54.187,175.501,16.034,152.327
C04917=1094.553,-4.810,-54.201,175.503,16.036,152.327
C04918=1094.560,-4.561,-54.214,175.505,16.037,152.327
C04919=1094.565,-4.311,-54.228,175.507,16.038,152.327
C04920=1094.571,-4.062,-54.241,175.508,16.039,152.327
C04921=1094.577,-3.812,-54.255,175.510,16.040,152.327
C04922=1094.583,-3.562,-54.267,175.513,16.042,152.326
C04923=1094.589,-3.312,-54.282,175.514,16.043,152.326
C04924=1094.594,-3.063,-54.295,175.516,16.044,152.326
C04925=1094.600,-2.813,-54.309,175.518,16.045,152.326
C04926=1094.606,-2.564,-54.323,175.519,16.046,152.326
C04927=1094.611,-2.314,-54.336,175.522,16.048,152.326
C04928=1094.618,-2.065,-54.350,175.523,16.049,152.325
C04929=1094.623,-1.815,-54.364,175.525,16.050,152.325
C04930=1094.629,-1.566,-54.377,175.527,16.051,152.325
C04931=1094.634,-1.316,-54.391,175.529,16.052,152.325
C04932=1094.640,-1.067,-54.405,175.531,16.053,152.325
C04933=1094.646,-0.796,-54.419,175.533,16.054,152.325
C04934=1094.653,-0.524,-54.434,175.535,16.056,152.324
C04935=1094.659,-0.253,-54.449,175.537,16.057,152.324
C04936=1094.665,0.019,-54.464,175.538,16.058,152.324
C04937=1094.671,0.269,-54.478,175.541,16.060,152.324
C04938=1094.676,0.518,-54.492,175.543,16.061,152.324
C04939=1094.682,0.768,-54.506,175.544,16.062,152.324
C04940=1094.688,1.017,-54.519,175.546,16.063,152.324
C04941=1094.693,1.267,-54.533,175.549,16.064,152.323
C04942=1094.699,1.516,-54.547,175.550,16.065,152.323
C04943=1094.704,1.766,-54.561,175.552,16.066,152.323
C04944=1094.711,2.015,-54.574,175.554,16.067,152.323
C04945=1094.717,2.265,-54.588,175.556,16.069,152.323
C04946=1094.722,2.515,-54.602,175.558,16.070,152.323
C04947=1094.728,2.765,-54.616,175.560,16.071,152.322
C04948=1094.734,3.014,-54.629,175.561,16.072,152.322
C04949=1094.740,3.263,-54.644,175.563,16.073,152.322
C04950=1094.745,3.512,-54.658,175.565,16.074,152.322
C04951=1094.751,3.762,-54.672,175.567,16.076,152.322
C04952=1094.757,4.012,-54.686,175.569,16.077,152.322
C04953=1094.763,4.261,-54.699,175.570,16.077,152.322
C04954=1094.768,4.511,-54.713,175.573,16.079,152.321
C04955=1094.774,4.761,-54.727,175.574,16.080,152.321
C04956=1094.779,5.010,-54.741,175.576,16.081,152.321
C04957=1094.786,5.260,-54.756,175.578,16.082,152.321
C04958=1094.791,5.509,-54.770,175.580,16.084,152.321
C04959=1094.797,5.759,-54.783,175.582,16.085,152.321
C04960=1094.803,6.008,-54.797,175.584,16.086,152.320
C04961=1094.808,6.258,-54.811,175.586,16.086,152.320
C04962=1094.815,6.508,-54.826,175.588,16.088,152.320
C04963=1094.820,6.757,-54.839,175.590,16.089,152.320
C04964=1094.826,7.007,-54.853,175.592,16.090,152.320
C04965=1094.832,7.256,-54.867,175.593,16.091,152.320
C04966=1094.837,7.505,-54.880,175.596,16.093,152.319
C04967=1094.844,7.755,-54.895,175.598,16.094,152.319
C04968=1094.849,8.005,-54.909,175.599,16.095,152.319
C04969=1094.855,8.254,-54.923,175.601,16.096,152.319
C04970=1094.860,8.504,-54.937,175.603,16.097,152.319
C04971=1094.867,8.754,-54.952,175.605,16.098,152.319
C04972=1094.873,9.003,-54.965,175.607,16.099,152.318
C04973=1094.878,9.252,-54.979,175.608,16.100,152.318
C04974=1094.884,9.501,-54.994,175.611,16.102,152.318
C04975=1094.890,9.752,-55.008,175.613,16.103,152.318
C04976=1094.896,10.001,-55.022,175.615,16.103,152.318
C04977=1094.901,10.250,-55.036,175.616,16.105,152.318
C04978=1094.907,10.500,-55.051,175.619,16.106,152.317
C04979=1094.913,10.750,-55.064,175.621,16.107,152.317
C04980=1094.919,10.999,-55.078,175.622,16.108,152.317
C04981=1094.925,11.248,-55.092,175.624,16.109,152.317
C04982=1094.931,11.498,-55.106,175.626,16.111,152.317
C04983=1094.937,11.747,-55.121,175.628,16.111,152.316
C04984=1094.942,11.997,-55.135,175.630,16.112,152.316
C04985=1094.948,12.247,-55.149,175.632,16.114,152.316
C04986=1094.954,12.496,-55.164,175.634,16.115,152.316
C04987=1094.960,12.746,-55.178,175.636,16.116,152.316
C04988=1094.966,12.995,-55.193,175.638,16.117,152.316
C04989=1094.971,13.245,-55.206,175.639,16.118,152.316
C04990=1094.977,13.495,-55.220,175.642,16.119,152.315
C04991=1094.983,13.744,-55.235,175.644,16.120,152.315
C04992=1094.989,13.994,-55.249,175.645,16.121,152.315
C04993=1094.995,14.243,-55.263,175.648,16.123,152.315
C04994=1095.001,14.493,-55.277,175.650,16.123,152.314
C04995=1095.006,14.742,-55.292,175.651,16.125,152.314
C04996=1095.012,14.992,-55.306,175.653,16.125,152.314
C04997=1095.018,15.265,-55.322,175.656,16.127,152.314
C04998=1095.024,15.538,-55.337,175.658,16.128,152.314
C04999=1095.031,15.812,-55.354,175.660,16.129,152.314
C05000=1095.038,16.085,-55.370,175.662,16.131,152.314
C05001=1095.043,16.335,-55.384,175.664,16.132,152.313
C05002=1095.049,16.584,-55.398,175.666,16.133,152.313
C05003=1095.055,16.834,-55.412,175.668,16.134,152.313
C05004=1095.061,17.083,-55.427,175.670,16.135,152.313
C05005=1095.066,17.333,-55.441,175.672,16.136,152.312
C05006=1095.072,17.583,-55.456,175.674,16.137,152.312
C05007=1095.077,17.832,-55.470,175.676,16.138,152.312
C05008=1095.084,18.082,-55.485,175.678,16.140,152.312
C05009=1095.089,18.331,-55.500,175.680,16.140,152.312
C05010=1095.095,18.580,-55.514,175.681,16.142,152.312
C05011=1095.101,18.830,-55.529,175.684,16.143,152.311
C05012=1095.107,19.080,-55.542,175.686,16.144,152.311
C05013=1095.112,19.329,-55.558,175.688,16.145,152.311
C05014=1095.118,19.578,-55.573,175.689,16.146,152.311
C05015=1095.124,19.828,-55.586,175.692,16.147,152.311
C05016=1095.130,20.078,-55.601,175.693,16.148,152.311
C05017=1095.136,20.327,-55.615,175.695,16.149,152.310
C05018=1095.141,20.576,-55.630,175.698,16.151,152.310
C05019=1095.147,20.826,-55.645,175.700,16.151,152.310
C05020=1095.152,21.076,-55.659,175.701,16.153,152.310
C05021=1095.158,21.325,-55.674,175.704,16.154,152.310
C05022=1095.165,21.574,-55.689,175.706,16.155,152.309
C05023=1095.169,21.824,-55.703,175.707,16.156,152.309
C05024=1095.176,22.074,-55.718,175.709,16.157,152.309
C05025=1095.181,22.323,-55.733,175.711,16.159,152.309
C05026=1095.187,22.572,-55.747,175.713,16.159,152.309
C05027=1095.193,22.822,-55.762,175.715,16.160,152.308
C05028=1095.198,23.071,-55.777,175.718,16.162,152.308
C05029=1095.205,23.321,-55.792,175.720,16.162,152.308
C05030=1095.209,23.571,-55.806,175.721,16.164,152.308
C05031=1095.215,23.820,-55.821,175.724,16.165,152.308
C05032=1095.222,24.070,-55.836,175.725,16.166,152.308
C05033=1095.227,24.318,-55.850,175.727,16.167,152.307
C05034=1095.233,24.569,-55.865,175.730,16.168,152.307
C05035=1095.239,24.818,-55.880,175.732,16.169,152.307
C05036=1095.245,25.068,-55.895,175.733,16.170,152.307
C05037=1095.250,25.317,-55.910,175.735,16.171,152.307
C05038=1095.256,25.567,-55.924,175.737,16.173,152.306
C05039=1095.262,25.816,-55.939,175.739,16.173,152.306
C05040=1095.267,26.065,-55.954,175.741,16.174,152.306
C05041=1095.273,26.315,-55.969,175.744,16.176,152.306
C05042=1095.279,26.564,-55.983,175.746,16.176,152.306
C05043=1095.285,26.814,-55.999,175.747,16.178,152.305
C05044=1095.290,27.064,-56.013,175.750,16.179,152.305
C05045=1095.297,27.313,-56.028,175.752,16.180,152.305
C05046=1095.302,27.563,-56.043,175.753,16.181,152.305
C05047=1095.308,27.812,-56.058,175.756,16.182,152.305
C05048=1095.314,28.061,-56.072,175.758,16.183,152.304
C05049=1095.319,28.311,-56.088,175.759,16.184,152.304
C05050=1095.325,28.560,-56.102,175.762,16.185,152.304
C05051=1095.331,28.810,-56.118,175.764,16.186,152.304
C05052=1095.336,29.060,-56.132,175.766,16.187,152.304
C05053=1095.343,29.309,-56.147,175.768,16.189,152.303
C05054=1095.348,29.559,-56.162,175.770,16.189,152.303
C05055=1095.354,29.808,-56.177,175.772,16.191,152.303
C05056=1095.359,30.057,-56.192,175.774,16.192,152.303
C05057=1095.366,30.307,-56.207,175.776,16.193,152.303
C05058=1095.371,30.556,-56.222,175.778,16.194,152.302
C05059=1095.377,30.806,-56.237,175.780,16.195,152.302
C05060=1095.382,31.055,-56.252,175.782,16.196,152.302
C05061=1095.389,31.331,-56.269,175.785,16.197,152.302
C05062=1095.395,31.605,-56.286,175.787,16.198,152.302
C05063=1095.401,31.880,-56.302,175.789,16.200,152.301
C05064=1095.407,32.155,-56.318,175.791,16.201,152.301
C05065=1095.414,32.405,-56.333,175.794,16.202,152.301
C05066=1095.419,32.654,-56.349,175.795,16.203,152.301
C05067=1095.425,32.903,-56.364,175.797,16.204,152.301
C05068=1095.430,33.152,-56.379,175.800,16.205,152.300
C05069=1095.436,33.402,-56.395,175.801,16.206,152.300
C05070=1095.442,33.651,-56.409,175.803,16.207,152.300
C05071=1095.447,33.901,-56.425,175.806,16.208,152.300
C05072=1095.453,34.150,-56.440,175.808,16.209,152.300
C05073=1095.459,34.400,-56.455,175.809,16.210,152.299
C05074=1095.465,34.650,-56.470,175.812,16.211,152.299
C05075=1095.470,34.899,-56.485,175.814,16.212,152.299
C05076=1095.477,35.149,-56.500,175.816,16.213,152.299
C05077=1095.482,35.398,-56.515,175.818,16.214,152.298
C05078=1095.488,35.648,-56.530,175.820,16.215,152.298
C05079=1095.493,35.896,-56.546,175.822,16.216,152.298
C05080=1095.499,36.146,-56.562,175.825,16.217,152.298
C05081=1095.505,36.396,-56.577,175.826,16.218,152.297
C05082=1095.510,36.645,-56.592,175.829,16.220,152.297
C05083=1095.517,36.895,-56.607,175.831,16.221,152.297
C05084=1095.522,37.144,-56.622,175.833,16.221,152.297
C05085=1095.528,37.393,-56.638,175.835,16.222,152.297
C05086=1095.534,37.643,-56.653,175.837,16.224,152.296
C05087=1095.539,37.892,-56.668,175.839,16.224,152.296
C05088=1095.546,38.142,-56.683,175.841,16.226,152.296
C05089=1095.551,38.392,-56.699,175.843,16.227,152.296
C05090=1095.557,38.641,-56.715,175.845,16.227,152.296
C05091=1095.562,38.891,-56.730,175.848,16.229,152.295
C05092=1095.568,39.139,-56.745,175.849,16.230,152.295
C05093=1095.574,39.389,-56.760,175.852,16.231,152.295
C05094=1095.580,39.639,-56.777,175.854,16.232,152.295
C05095=1095.585,39.888,-56.792,175.856,16.233,152.294
C05096=1095.591,40.138,-56.807,175.858,16.234,152.294
C05097=1095.596,40.387,-56.822,175.860,16.235,152.294
C05098=1095.602,40.636,-56.838,175.862,16.236,152.294
C05099=1095.608,40.886,-56.854,175.865,16.237,152.294
C05100=1095.614,41.135,-56.868,175.866,16.238,152.293
C05101=1095.619,41.385,-56.884,175.869,16.239,152.293
C05102=1095.625,41.635,-56.900,175.871,16.240,152.293
C05103=1095.630,41.884,-56.915,175.873,16.241,152.293
C05104=1095.637,42.134,-56.930,175.875,16.242,152.292
C05105=1095.642,42.383,-56.947,175.877,16.243,152.292
C05106=1095.648,42.632,-56.962,175.879,16.244,152.292
C05107=1095.653,42.881,-56.978,175.882,16.245,152.292
C05108=1095.659,43.131,-56.994,175.883,16.246,152.291
C05109=1095.665,43.380,-57.008,175.886,16.248,152.291
C05110=1095.671,43.630,-57.024,175.888,16.248,152.291
C05111=1095.677,43.880,-57.040,175.890,16.249,152.291
C05112=1095.682,44.129,-57.055,175.892,16.250,152.291
C05113=1095.687,44.378,-57.071,175.894,16.251,152.290
C05114=1095.693,44.628,-57.087,175.896,16.252,152.290
C05115=1095.698,44.877,-57.103,175.898,16.253,152.290
C05116=1095.704,45.127,-57.118,175.900,16.254,152.290
C05117=1095.709,45.376,-57.134,175.903,16.255,152.289
C05118=1095.715,45.626,-57.150,175.905,16.256,152.289
C05119=1095.721,45.875,-57.165,175.907,16.257,152.289
C05120=1095.726,46.124,-57.181,175.909,16.258,152.289
C05121=1095.732,46.374,-57.197,175.911,16.259,152.289
C05122=1095.738,46.623,-57.213,175.914,16.261,152.288
C05123=1095.743,46.873,-57.228,175.915,16.262,152.288
C05124=1095.749,47.122,-57.244,175.917,16.262,152.288
C05125=1095.756,47.397,-57.262,175.920,16.263,152.288
C05126=1095.762,47.672,-57.279,175.923,16.265,152.287
C05127=1095.767,47.947,-57.296,175.925,16.265,152.287
C05128=1095.774,48.222,-57.313,175.927,16.267,152.287
C05129=1095.780,48.471,-57.330,175.929,16.267,152.287
C05130=1095.785,48.721,-57.345,175.932,16.269,152.286
C05131=1095.791,48.970,-57.361,175.933,16.270,152.286
C05132=1095.796,49.219,-57.377,175.936,16.271,152.286
C05133=1095.802,49.469,-57.393,175.938,16.272,152.286
C05134=1095.807,49.718,-57.409,175.940,16.272,152.285
C05135=1095.813,49.968,-57.424,175.943,16.274,152.285
C05136=1095.819,50.217,-57.441,175.944,16.274,152.285
C05137=1095.825,50.467,-57.456,175.947,16.276,152.285
C05138=1095.831,50.716,-57.472,175.949,16.277,152.284
C05139=1095.836,50.965,-57.488,175.951,16.278,152.284
C05140=1095.842,51.215,-57.504,175.953,16.279,152.284
C05141=1095.848,51.464,-57.520,175.955,16.280,152.284
C05142=1095.854,51.714,-57.536,175.958,16.281,152.283
C05143=1095.859,51.963,-57.552,175.960,16.281,152.283
C05144=1095.865,52.212,-57.568,175.963,16.283,152.283
C05145=1095.870,52.462,-57.584,175.964,16.283,152.283
C05146=1095.876,52.712,-57.600,175.966,16.284,152.282
C05147=1095.882,52.961,-57.616,175.969,16.285,152.282
C05148=1095.887,53.210,-57.632,175.971,16.286,152.282
C05149=1095.892,53.460,-57.648,175.974,16.287,152.282
C05150=1095.898,53.709,-57.664,175.975,16.288,152.281
C05151=1095.904,53.959,-57.680,175.977,16.289,152.281
C05152=1095.910,54.208,-57.697,175.980,16.290,152.281
C05153=1095.915,54.457,-57.712,175.982,16.291,152.281
C05154=1095.921,54.707,-57.728,175.985,16.292,152.280
C05155=1095.927,54.956,-57.744,175.987,16.293,152.280
C05156=1095.933,55.205,-57.761,175.989,16.294,152.280
C05157=1095.939,55.455,-57.776,175.991,16.295,152.279
C05158=1095.945,55.705,-57.792,175.993,16.295,152.279
C05159=1095.950,55.954,-57.809,175.996,16.297,152.279
C05160=1095.955,56.203,-57.825,175.998,16.297,152.279
C05161=1095.961,56.452,-57.841,176.000,16.299,152.278
C05162=1095.967,56.702,-57.858,176.002,16.299,152.278
C05163=1095.973,56.952,-57.873,176.004,16.300,152.278
C05164=1095.979,57.201,-57.889,176.007,16.301,152.278
C05165=1095.985,57.450,-57.906,176.009,16.302,152.277
C05166=1095.990,57.700,-57.923,176.011,16.303,152.277
C05167=1095.996,57.949,-57.939,176.013,16.304,152.277
C05168=1096.002,58.199,-57.955,176.016,16.305,152.277
C05169=1096.008,58.448,-57.971,176.018,16.306,152.276
C05170=1096.013,58.697,-57.987,176.020,16.306,152.276
C05171=1096.019,58.947,-58.003,176.023,16.307,152.276
C05172=1096.024,59.196,-58.020,176.025,16.308,152.275
C05173=1096.030,59.446,-58.036,176.027,16.309,152.275
C05174=1096.036,59.695,-58.052,176.029,16.310,152.275
C05175=1096.042,59.944,-58.068,176.032,16.311,152.275
C05176=1096.048,60.194,-58.085,176.034,16.312,152.274
C05177=1096.054,60.443,-58.101,176.036,16.313,152.274
C05178=1096.059,60.693,-58.118,176.038,16.314,152.274
C05179=1096.065,60.942,-58.134,176.040,16.314,152.273
C05180=1096.071,61.191,-58.150,176.043,16.315,152.273
C05181=1096.077,61.441,-58.167,176.045,16.316,152.273
C05182=1096.083,61.690,-58.183,176.048,16.317,152.273
C05183=1096.088,61.940,-58.200,176.050,16.318,152.272
C05184=1096.094,62.189,-58.216,176.053,16.319,152.272
C05185=1096.100,62.438,-58.232,176.055,16.319,152.272
C05186=1096.106,62.688,-58.248,176.056,16.320,152.271
C05187=1096.111,62.937,-58.265,176.059,16.321,152.271
C05188=1096.117,63.187,-58.282,176.061,16.322,152.271
C05189=1096.123,63.461,-58.300,176.064,16.323,152.270
C05190=1096.130,63.736,-58.317,176.067,16.324,152.270
C05191=1096.137,64.011,-58.336,176.069,16.325,152.270
C05192=1096.143,64.285,-58.354,176.072,16.326,152.269
C05193=1096.149,64.534,-58.371,176.073,16.326,152.269
C05194=1096.154,64.784,-58.388,176.076,16.328,152.269
C05195=1096.160,65.033,-58.404,176.078,16.328,152.269
C05196=1096.166,65.283,-58.420,176.081,16.329,152.268
C05197=1096.171,65.532,-58.437,176.083,16.330,152.268
C05198=1096.177,65.782,-58.453,176.086,16.331,152.268
C05199=1096.182,66.031,-58.470,176.087,16.332,152.267
C05200=1096.189,66.280,-58.487,176.090,16.333,152.267
C05201=1096.195,66.530,-58.503,176.092,16.333,152.267
C05202=1096.200,66.779,-58.520,176.095,16.335,152.267
C05203=1096.206,67.029,-58.536,176.097,16.335,152.266
C05204=1096.211,67.278,-58.553,176.100,16.337,152.266
C05205=1096.217,67.527,-58.570,176.102,16.337,152.266
C05206=1096.222,67.777,-58.587,176.104,16.337,152.265
C05207=1096.228,68.026,-58.603,176.106,16.339,152.265
C05208=1096.234,68.276,-58.620,176.108,16.339,152.265
C05209=1096.240,68.525,-58.636,176.111,16.340,152.264
C05210=1096.245,68.774,-58.654,176.113,16.341,152.264
C05211=1096.251,69.023,-58.670,176.116,16.342,152.264
C05212=1096.257,69.273,-58.687,176.118,16.342,152.263
C05213=1096.262,69.522,-58.703,176.121,16.344,152.263
C05214=1096.268,69.771,-58.720,176.123,16.344,152.263
C05215=1096.274,70.021,-58.737,176.125,16.346,152.263
C05216=1096.279,70.270,-58.754,176.127,16.346,152.262
C05217=1096.285,70.519,-58.771,176.130,16.347,152.262
C05218=1096.290,70.769,-58.788,176.132,16.348,152.262
C05219=1096.296,71.018,-58.804,176.134,16.348,152.261
C05220=1096.302,71.267,-58.822,176.137,16.349,152.261
C05221=1096.308,71.516,-58.838,176.139,16.350,152.261
C05222=1096.313,71.766,-58.855,176.142,16.351,152.260
C05223=1096.318,72.015,-58.872,176.144,16.352,152.260
C05224=1096.325,72.265,-58.889,176.146,16.353,152.260
C05225=1096.330,72.515,-58.906,176.149,16.353,152.259
C05226=1096.336,72.764,-58.923,176.151,16.354,152.259
C05227=1096.342,73.013,-58.940,176.153,16.355,152.259
C05228=1096.347,73.263,-58.956,176.156,16.356,152.258
C05229=1096.353,73.512,-58.973,176.158,16.357,152.258
C05230=1096.358,73.761,-58.990,176.161,16.358,152.258
C05231=1096.364,74.010,-59.008,176.163,16.358,152.258
C05232=1096.370,74.260,-59.024,176.166,16.359,152.257
C05233=1096.375,74.509,-59.042,176.167,16.360,152.257
C05234=1096.381,74.758,-59.059,176.170,16.361,152.257
C05235=1096.387,75.008,-59.076,176.172,16.361,152.256
C05236=1096.393,75.258,-59.093,176.175,16.362,152.256
C05237=1096.398,75.507,-59.110,176.177,16.363,152.256
C05238=1096.404,75.756,-59.127,176.180,16.364,152.255
C05239=1096.409,76.006,-59.143,176.182,16.364,152.255
C05240=1096.415,76.255,-59.161,176.185,16.366,152.255
C05241=1096.421,76.503,-59.178,176.187,16.366,152.254
C05242=1096.427,76.754,-59.195,176.190,16.367,152.254
C05243=1096.432,77.003,-59.213,176.192,16.367,152.254
C05244=1096.438,77.252,-59.229,176.194,16.368,152.253
C05245=1096.444,77.501,-59.247,176.197,16.369,152.253
C05246=1096.449,77.751,-59.263,176.199,16.370,152.253
C05247=1096.455,78.000,-59.281,176.202,16.370,152.252
C05248=1096.461,78.250,-59.298,176.203,16.371,152.252
C05249=1096.467,78.499,-59.315,176.206,16.372,152.252
C05250=1096.472,78.748,-59.333,176.208,16.373,152.251
C05251=1096.477,78.998,-59.350,176.211,16.374,152.251
C05252=1096.484,79.246,-59.367,176.213,16.374,152.251
C05253=1096.489,79.521,-59.386,176.216,16.375,152.250
C05254=1096.496,79.796,-59.405,176.219,16.376,152.250
C05255=1096.502,80.071,-59.424,176.222,16.377,152.249
C05256=1096.509,80.345,-59.443,176.224,16.378,152.249
C05257=1096.514,80.595,-59.460,176.227,16.379,152.249
C05258=1096.519,80.844,-59.478,176.229,16.379,152.249
C05259=1096.525,81.093,-59.495,176.232,16.380,152.248
C05260=1096.530,81.342,-59.512,176.233,16.381,152.248
C05261=1096.536,81.592,-59.530,176.236,16.382,152.247
C05262=1096.542,81.841,-59.547,176.238,16.382,152.247
C05263=1096.548,82.091,-59.564,176.241,16.383,152.247
C05264=1096.553,82.340,-59.581,176.243,16.384,152.247
C05265=1096.559,82.589,-59.599,176.246,16.385,152.246
C05266=1096.565,82.838,-59.617,176.249,16.385,152.246
C05267=1096.570,83.088,-59.634,176.251,16.386,152.245
C05268=1096.576,83.337,-59.651,176.254,16.387,152.245
C05269=1096.581,83.586,-59.669,176.256,16.388,152.245
C05270=1096.587,83.836,-59.687,176.259,16.388,152.244
C05271=1096.592,84.086,-59.704,176.261,16.389,152.244
C05272=1096.598,84.335,-59.721,176.264,16.390,152.244
C05273=1096.603,84.584,-59.739,176.266,16.390,152.243
C05274=1096.610,84.833,-59.757,176.269,16.391,152.243
C05275=1096.615,85.082,-59.774,176.271,16.392,152.243
C05276=1096.621,85.331,-59.791,176.274,16.392,152.242
C05277=1096.627,85.581,-59.808,176.276,16.393,152.242
C05278=1096.633,85.831,-59.826,176.279,16.394,152.241
C05279=1096.638,86.080,-59.843,176.281,16.395,152.241
C05280=1096.644,86.329,-59.861,176.284,16.395,152.241
C05281=1096.650,86.578,-59.879,176.286,16.396,152.240
C05282=1096.655,86.827,-59.897,176.288,16.397,152.240
C05283=1096.661,87.076,-59.914,176.291,16.397,152.240
C05284=1096.667,87.326,-59.932,176.294,16.398,152.239
C05285=1096.672,87.576,-59.949,176.296,16.398,152.239
C05286=1096.678,87.825,-59.966,176.298,16.400,152.239
C05287=1096.684,88.075,-59.984,176.301,16.400,152.238
C05288=1096.689,88.324,-60.002,176.304,16.401,152.238
C05289=1096.695,88.573,-60.020,176.306,16.401,152.238
C05290=1096.701,88.822,-60.037,176.308,16.402,152.237
C05291=1096.707,89.071,-60.055,176.311,16.402,152.237
C05292=1096.712,89.320,-60.073,176.314,16.403,152.236
C05293=1096.718,89.570,-60.091,176.316,16.404,152.236
C05294=1096.724,89.819,-60.108,176.319,16.405,152.236
C05295=1096.729,90.068,-60.126,176.321,16.405,152.235
C05296=1096.735,90.318,-60.144,176.324,16.406,152.235
C05297=1096.741,90.567,-60.161,176.327,16.406,152.234
C05298=1096.746,90.817,-60.180,176.329,16.407,152.234
C05299=1096.752,91.066,-60.197,176.332,16.408,152.234
C05300=1096.757,91.315,-60.215,176.334,16.408,152.233
C05301=1096.763,91.565,-60.233,176.337,16.409,152.233
C05302=1096.769,91.814,-60.250,176.339,16.410,152.233
C05303=1096.775,92.062,-60.269,176.342,16.411,152.232
C05304=1096.780,92.312,-60.287,176.344,16.411,152.232
C05305=1096.786,92.562,-60.305,176.347,16.412,152.231
C05306=1096.791,92.811,-60.322,176.349,16.412,152.231
C05307=1096.797,93.060,-60.340,176.352,16.413,152.231
C05308=1096.803,93.309,-60.358,176.354,16.413,152.230
C05309=1096.808,93.559,-60.376,176.357,16.414,152.230
C05310=1096.814,93.808,-60.394,176.360,16.415,152.229
C05311=1096.819,94.057,-60.411,176.362,16.416,152.229
C05312=1096.826,94.307,-60.430,176.365,16.416,152.229
C05313=1096.830,94.556,-60.448,176.367,16.417,152.228
C05314=1096.836,94.805,-60.466,176.370,16.417,152.228
C05315=1096.842,95.055,-60.484,176.372,16.418,152.227
C05316=1096.848,95.304,-60.501,176.375,16.419,152.227
C05317=1096.854,95.579,-60.522,176.378,16.419,152.227
C05318=1096.860,95.853,-60.541,176.380,16.420,152.226
C05319=1096.867,96.128,-60.562,176.383,16.420,152.226
C05320=1096.873,96.402,-60.582,176.386,16.421,152.225
C05321=1096.879,96.652,-60.599,176.389,16.422,152.225
C05322=1096.883,96.901,-60.618,176.391,16.422,152.225
C05323=1096.889,97.150,-60.635,176.394,16.423,152.224
C05324=1096.895,97.399,-60.654,176.396,16.423,152.224
C05325=1096.901,97.648,-60.671,176.399,16.424,152.223
C05326=1096.906,97.898,-60.690,176.401,16.425,152.223
C05327=1096.912,98.147,-60.708,176.404,16.426,152.223
C05328=1096.918,98.396,-60.726,176.406,16.426,152.222
C05329=1096.923,98.646,-60.744,176.409,16.427,152.222
C05330=1096.929,98.895,-60.763,176.412,16.427,152.221
C05331=1096.935,99.144,-60.781,176.415,16.428,152.221
C05332=1096.940,99.394,-60.799,176.417,16.429,152.220
C05333=1096.946,99.642,-60.817,176.420,16.429,152.220
C05334=1096.952,99.892,-60.835,176.423,16.430,152.220
C05335=1096.957,100.142,-60.853,176.425,16.430,152.219
C05336=1096.963,100.391,-60.872,176.428,16.431,152.219
C05337=1096.969,100.640,-60.890,176.430,16.431,152.218
C05338=1096.975,100.889,-60.909,176.433,16.432,152.218
C05339=1096.980,101.138,-60.926,176.435,16.432,152.218
C05340=1096.986,101.388,-60.944,176.438,16.432,152.217
C05341=1096.991,101.637,-60.963,176.441,16.434,152.217
C05342=1096.998,101.886,-60.981,176.443,16.434,152.216
C05343=1097.003,102.135,-61.000,176.446,16.435,152.216
C05344=1097.009,102.385,-61.018,176.448,16.435,152.216
C05345=1097.014,102.634,-61.037,176.451,16.436,152.215
C05346=1097.020,102.883,-61.055,176.454,16.436,152.215
C05347=1097.025,103.132,-61.074,176.457,16.436,152.214
C05348=1097.031,103.382,-61.092,176.460,16.437,152.214
C05349=1097.036,103.631,-61.111,176.462,16.437,152.213
C05350=1097.042,103.880,-61.128,176.465,16.438,152.213
C05351=1097.048,104.130,-61.148,176.467,16.438,152.212
C05352=1097.053,104.379,-61.166,176.470,16.439,152.212
C05353=1097.059,104.628,-61.184,176.472,16.439,152.212
C05354=1097.064,104.878,-61.203,176.475,16.440,152.211
C05355=1097.070,105.127,-61.221,176.478,16.441,152.211
C05356=1097.075,105.376,-61.239,176.480,16.441,152.210
C05357=1097.082,105.625,-61.258,176.483,16.442,152.210
C05358=1097.087,105.874,-61.277,176.486,16.442,152.210
C05359=1097.093,106.124,-61.295,176.489,16.443,152.209
C05360=1097.099,106.373,-61.314,176.491,16.443,152.209
C05361=1097.103,106.622,-61.332,176.494,16.444,152.208
C05362=1097.110,106.872,-61.351,176.497,16.445,152.208
C05363=1097.115,107.120,-61.370,176.499,16.445,152.207
C05364=1097.121,107.370,-61.388,176.502,16.446,152.207
C05365=1097.127,107.619,-61.407,176.504,16.446,152.206
C05366=1097.132,107.868,-61.425,176.508,16.446,152.206
C05367=1097.138,108.118,-61.444,176.511,16.447,152.205
C05368=1097.143,108.367,-61.463,176.513,16.447,152.205
C05369=1097.149,108.616,-61.481,176.516,16.448,152.205
C05370=1097.155,108.866,-61.500,176.518,16.448,152.204
C05371=1097.161,109.114,-61.518,176.521,16.449,152.204
C05372=1097.166,109.364,-61.537,176.523,16.449,152.203
C05373=1097.172,109.613,-61.557,176.526,16.450,152.203
C05374=1097.177,109.862,-61.574,176.529,16.451,152.202
C05375=1097.183,110.112,-61.593,176.532,16.450,152.202
C05376=1097.189,110.361,-61.613,176.535,16.451,152.201
C05377=1097.195,110.609,-61.631,176.537,16.451,152.201
C05378=1097.200,110.859,-61.650,176.540,16.452,152.200
C05379=1097.206,111.109,-61.669,176.543,16.453,152.200
C05380=1097.212,111.357,-61.687,176.545,16.453,152.200
C05381=1097.217,111.633,-61.708,176.549,16.453,152.199
C05382=1097.224,111.907,-61.729,176.552,16.454,152.199
C05383=1097.230,112.182,-61.750,176.555,16.454,152.198
C05384=1097.237,112.456,-61.771,176.558,16.455,152.198
C05385=1097.242,112.705,-61.790,176.560,16.455,152.197
C05386=1097.248,112.954,-61.809,176.563,16.456,152.197
C05387=1097.254,113.204,-61.827,176.566,16.456,152.196
C05388=1097.259,113.453,-61.846,176.569,16.456,152.196
C05389=1097.265,113.702,-61.865,176.572,16.457,152.195
C05390=1097.270,113.952,-61.884,176.574,16.458,152.195
C05391=1097.277,114.201,-61.903,176.577,16.458,152.194
C05392=1097.282,114.450,-61.922,176.579,16.458,152.194
C05393=1097.287,114.699,-61.941,176.582,16.459,152.193
C05394=1097.293,114.948,-61.960,176.586,16.459,152.193
C05395=1097.298,115.197,-61.979,176.588,16.460,152.192
C05396=1097.304,115.447,-61.998,176.591,16.460,152.192
C05397=1097.310,115.696,-62.017,176.593,16.461,152.192
C05398=1097.315,115.945,-62.036,176.596,16.461,152.191
C05399=1097.320,116.194,-62.056,176.599,16.462,152.191
C05400=1097.326,116.444,-62.075,176.601,16.462,152.190
C05401=1097.331,116.692,-62.094,176.605,16.462,152.190
C05402=1097.338,116.942,-62.112,176.607,16.463,152.189
C05403=1097.343,117.191,-62.132,176.610,16.463,152.189
C05404=1097.349,117.440,-62.151,176.613,16.464,152.188
C05405=1097.354,117.689,-62.170,176.615,16.464,152.188
C05406=1097.360,117.939,-62.189,176.618,16.464,152.187
C05407=1097.365,118.188,-62.208,176.621,16.465,152.187
C05408=1097.371,118.437,-62.227,176.624,16.466,152.186
C05409=1097.376,118.686,-62.246,176.627,16.466,152.186
C05410=1097.382,118.936,-62.266,176.629,16.466,152.185
C05411=1097.388,119.185,-62.285,176.632,16.467,152.185
C05412=1097.393,119.434,-62.304,176.635,16.467,152.184
C05413=1097.398,119.683,-62.323,176.638,16.467,152.184
C05414=1097.404,119.933,-62.342,176.641,16.468,152.183
C05415=1097.410,120.181,-62.362,176.643,16.468,152.183
C05416=1097.416,120.431,-62.381,176.646,16.469,152.183
C05417=1097.421,120.680,-62.400,176.649,16.469,152.182
C05418=1097.426,120.929,-62.419,176.652,16.469,152.182
C05419=1097.432,121.178,-62.439,176.655,16.470,152.181
C05420=1097.438,121.428,-62.458,176.657,16.470,152.181
C05421=1097.444,121.677,-62.478,176.660,16.470,152.180
C05422=1097.449,121.925,-62.497,176.663,16.471,152.180
C05423=1097.455,122.175,-62.516,176.666,16.471,152.179
C05424=1097.460,122.424,-62.535,176.669,16.472,152.179
C05425=1097.466,122.673,-62.556,176.672,16.472,152.178
C05426=1097.471,122.923,-62.575,176.674,16.472,152.178
C05427=1097.477,123.172,-62.594,176.678,16.473,152.177
C05428=1097.483,123.422,-62.614,176.680,16.473,152.177
C05429=1097.488,123.670,-62.633,176.683,16.473,152.176
C05430=1097.494,123.919,-62.652,176.686,16.474,152.175
C05431=1097.499,124.169,-62.672,176.688,16.474,152.175
C05432=1097.505,124.418,-62.692,176.692,16.474,152.174
C05433=1097.511,124.667,-62.711,176.695,16.475,152.174
C05434=1097.517,124.916,-62.730,176.697,16.475,152.174
C05435=1097.523,125.165,-62.750,176.700,16.475,152.173
C05436=1097.528,125.415,-62.769,176.703,16.476,152.173
C05437=1097.534,125.663,-62.788,176.706,16.476,152.172
C05438=1097.539,125.912,-62.809,176.709,16.476,152.171
C05439=1097.544,126.162,-62.828,176.711,16.476,152.171
C05440=1097.550,126.411,-62.847,176.715,16.477,152.170
C05441=1097.556,126.660,-62.867,176.718,16.477,152.170
C05442=1097.562,126.910,-62.886,176.720,16.477,152.169
C05443=1097.568,127.158,-62.906,176.723,16.478,152.169
C05444=1097.574,127.408,-62.926,176.726,16.478,152.168
C05445=1097.580,127.682,-62.947,176.729,16.478,152.168
C05446=1097.586,127.957,-62.969,176.732,16.478,152.167
C05447=1097.592,128.232,-62.990,176.735,16.479,152.167
C05448=1097.599,128.507,-63.012,176.739,16.479,152.166
C05449=1097.605,128.756,-63.032,176.742,16.479,152.165
C05450=1097.610,129.004,-63.051,176.744,16.479,152.165
C05451=1097.615,129.254,-63.072,176.747,16.480,152.164
C05452=1097.621,129.502,-63.092,176.751,16.480,152.164
